//Storage Area Service
RegisterAlarm(Trigger := fbStorageArea.fbWarehouse.fbReloadBox.Error,				ID := GVL_ErrorCode.GC_ALARM_STO_RELOAD_BOX,value := E_Severity.Level4,Message := fbStorageArea.fbWarehouse.fbReloadBox.Status,			Category := 1);
RegisterAlarm(Trigger := fbStorageArea.fbWarehouse.fbFeedInBox.Error,				ID := GVL_ErrorCode.GC_ALARM_STO_FEEDIN_BOX,value := E_Severity.Level4,Message := fbStorageArea.fbWarehouse.fbFeedInBox.Status,			Category := 1);
RegisterAlarm(Trigger := fbStorageArea.fbAddBoxes.Error ,							ID := GVL_ErrorCode.GC_ALARM_STO_ADD_BOXES,value := E_Severity.Level4,Message := fbStorageArea.fbAddBoxes.Status,							Category := 1);
RegisterAlarm(Trigger := fbStorageArea.fbBoxSupplyCtrl.Error ,						ID := GVL_ErrorCode.GC_ALARM_STO_BOX_SUPPLY,value := E_Severity.Level4,Message := fbStorageArea.fbBoxSupplyCtrl.Status,					Category := 1);
RegisterAlarm(Trigger := fbStorageArea.fbFeedInEmptyBoxWithRobot.Error ,			ID := GVL_ErrorCode.GC_ALARM_STO_FEEDIN_EMPTY,value := E_Severity.Level4,Message := fbStorageArea.fbFeedInEmptyBoxWithRobot.Status,			Category := 1);
RegisterAlarm(Trigger := fbStorageArea.fbReloadRoundBeltBoxWithRobot.Error ,		ID := GVL_ErrorCode.GC_ALARM_STO_RELOAD_ROUNDBELT,value := E_Severity.Level4,Message := fbStorageArea.fbReloadRoundBeltBoxWithRobot.Status,		Category := 1);
RegisterAlarm(Trigger := fbStorageArea.fbRobotAbsMove.Error ,						ID := GVL_ErrorCode.GC_ALARM_STO_ROBOT_ABS_MOVE,value := E_Severity.Level4,Message := fbStorageArea.fbRobotAbsMove.Status,						Category := 1);
RegisterAlarm(Trigger := fbStorageArea.fbRobotRegionMove_AllocatedConveyor.Error ,	ID := GVL_ErrorCode.GC_ALARM_STO_REGION_ALLOC_CV,value := E_Severity.Level4,Message := fbStorageArea.fbRobotRegionMove_AllocatedConveyor.Status,Category := 1);
RegisterAlarm(Trigger := fbStorageArea.fbRobotRegionMove_BufferArea.Error ,			ID := GVL_ErrorCode.GC_ALARM_STO_REGION_BUFFER,value := E_Severity.Level4,Message := fbStorageArea.fbRobotRegionMove_BufferArea.Status,		Category := 1);
RegisterAlarm(Trigger := fbStorageArea.fbRobotRegionMove_FeedInConveyor.Error ,		ID := GVL_ErrorCode.GC_ALARM_STO_REGION_FEEDIN_CV,value := E_Severity.Level4,Message := fbStorageArea.fbRobotRegionMove_FeedInConveyor.Status,	Category := 1);
RegisterAlarm(Trigger := fbStorageArea.fbRobotRegionMove_PullOutConveyor.Error ,	ID := GVL_ErrorCode.GC_ALARM_STO_REGION_PULLOUT_CV,value := E_Severity.Level4,Message := fbStorageArea.fbRobotRegionMove_PullOutConveyor.Status,	Category := 1);
RegisterAlarm(Trigger := fbStorageArea.fbRobotRegionMove_RoundBelt.Error ,			ID := GVL_ErrorCode.GC_ALARM_STO_REGION_ROUNDBELT,value := E_Severity.Level4,Message := fbStorageArea.fbRobotRegionMove_RoundBelt.Status,		Category := 1);
RegisterAlarm(Trigger := fbStorageArea.fbUpperFeedInConveyor.Error ,				ID := GVL_ErrorCode.GC_ALARM_STO_UPPER_FEEDIN_CV,value := E_Severity.Level4,Message := fbStorageArea.fbUpperFeedInConveyor.Status,				Category := 1);
RegisterAlarm(Trigger := fbStorageArea.fbWareHouseWithRobotMove.Error ,				ID := GVL_ErrorCode.GC_ALARM_STO_WAREHOUSE_ROBOT,value := E_Severity.Level4,Message := fbStorageArea.fbWareHouseWithRobotMove.Status,			Category := 1);



//Storage Cabinet Internal Service
RegisterAlarm(Trigger := fbStorageArea.fbFeedInRoundBeltBoxToWareHouse.Error,		ID := GVL_ErrorCode.GC_ALARM_STO_FEEDIN_RB_TO_WH,value := E_Severity.Level3,Message := fbStorageArea.fbFeedInRoundBeltBoxToWareHouse.Status,Category := 1);
RegisterAlarm(Trigger := fbStorageArea._fbDaimeterMovement.Error,					ID := GVL_ErrorCode.GC_ALARM_STO_DIAMETER_MOVEMENT,value := E_Severity.Level3,Message := fbStorageArea._fbDaimeterMovement.Status,			Category := 1);
RegisterAlarm(Trigger := fbStorageArea.fbRobotSelfHoming.Error,						ID := GVL_ErrorCode.GC_ALARM_STO_ROBOTSELFHOMING,value := E_Severity.Level3,Message := fbStorageArea.fbRobotSelfHoming.Status,				Category := 1);
RegisterAlarm(Trigger := fbStorageArea.fbWareHouseInnerPickToRoundBelt.Error,		ID := GVL_ErrorCode.GC_AlARM_STO_ROBOTINNERPICK,value := E_Severity.Level3,Message := fbStorageArea.fbWareHouseInnerPickToRoundBelt.Status,	Category := 1);
RegisterAlarm(Trigger := fbStorageArea.fbWareHouseInnerPickToRoundBeltBatch.Error,  ID := GVL_ErrorCode.GC_AlARM_STO_ROBOTINNERPICK_BATCH,value := E_Severity.Level3,Message := fbStorageArea.fbWareHouseInnerPickToRoundBeltBatch.Status,	Category := 1);
RegisterAlarm(Trigger := fbStorageArea.fbFeedInRoundBeltBoxBatch.Error,  			ID := GVL_ErrorCode.GC_AlARM_STO_ROUNDBELTTOWAREHOUSE_BATCH,value := E_Severity.Level3,Message := fbStorageArea.fbFeedInRoundBeltBoxBatch.Status,	Category := 1);


//Allocate Area Service
RegisterAlarm(Trigger := fbAllocateArea.fb_AllocateBatchMode.Error ,				ID := GVL_ErrorCode.GC_ALARM_ALC_BATCH_MODE,value := E_Severity.Level3,Message := fbAllocateArea.fb_AllocateBatchMode.Status,			Category := 2);
RegisterAlarm(Trigger := fbAllocateArea.fb_AllocateBatchMode_Reverse.Error ,		ID := GVL_ErrorCode.GC_ALARM_ALC_BATCH_REVERSE,value := E_Severity.Level3,Message := fbAllocateArea.fb_AllocateBatchMode_Reverse.Status,	Category := 2);
RegisterAlarm(Trigger := fbAllocateArea.fbDifferentCVCamera.xError ,				ID := GVL_ErrorCode.GC_ALARM_ALC_DIFF_CV_CAMERA,value := E_Severity.Level3,Message := fbAllocateArea.fbDifferentCVCamera.ErrorMsg,			Category := 2);
RegisterAlarm(Trigger := fbAllocateArea.fbOutRobot_BoxMoveReverse.Error ,			ID := GVL_ErrorCode.GC_ALARM_ALC_OUTROBOT_REVERSE,value := E_Severity.Level3,Message := fbAllocateArea.fbOutRobot_BoxMoveReverse.Status,		Category := 2);
RegisterAlarm(Trigger := fbAllocateArea.fbOutRobot_EmptyBoxMove.Error ,				ID := GVL_ErrorCode.GC_ALARM_ALC_OUTROBOT_EMPTY,value := E_Severity.Level3,Message := fbAllocateArea.fbOutRobot_EmptyBoxMove.Status,		Category := 2);
RegisterAlarm(Trigger := fbAllocateArea.fbOutRobot_RareBoxMove.Error ,				ID := GVL_ErrorCode.GC_ALARM_ALC_OUTROBOT_RARE,value := E_Severity.Level3,Message := fbAllocateArea.fbOutRobot_RareBoxMove.Status,		Category := 2);
RegisterAlarm(Trigger := fbAllocateArea.fbPulloutCV.Error ,							ID := GVL_ErrorCode.GC_ALARM_ALC_PULLOUT_CV,value := E_Severity.Level3,Message := fbAllocateArea.fbPulloutCV.Status,					Category := 2);
RegisterAlarm(Trigger := fbAllocateArea.RoundBeltControl.xError ,					ID := GVL_ErrorCode.GC_ALARM_ALC_ROUNDBELT,value := E_Severity.Level3,Message := fbAllocateArea.RoundBeltControl.ErrorMsg,			Category := 2);
RegisterAlarm(Trigger := fbAllocateArea.fbSameSizeCVCamera.xError ,					ID := GVL_ErrorCode.GC_ALARM_ALC_SAME_CV_CAMERA,value := E_Severity.Level3,Message := fbAllocateArea.fbSameSizeCVCamera.ErrorMsg,			Category := 2);
RegisterAlarm(Trigger := fbAllocateArea.fbSameSizeCVCamera_Reverse.xError ,			ID := GVL_ErrorCode.GC_ALARM_ALC_SAME_CV_CAMERA_REVERSE,value := E_Severity.Level3,Message := fbAllocateArea.fbSameSizeCVCamera_Reverse.ErrorMsg,	Category := 2);
RegisterAlarm(Trigger := fbAllocateArea.TurnTableControl.xError ,					ID := GVL_ErrorCode.GC_ALARM_ALC_TURNTABLE,value := E_Severity.Level3,Message := fbAllocateArea.TurnTableControl.ErrorMsg,			Category := 2);
RegisterAlarm(Trigger := fbAllocateArea.fbOutRobot_TurnTableToRoundBelt.Error ,		ID := GVL_ErrorCode.GC_ALARM_ALC_OUTROBOT_TT_TO_RB,value := E_Severity.Level3,Message := fbAllocateArea.fbOutRobot_TurnTableToRoundBelt.Status,Category := 2);
RegisterAlarm(Trigger := fbAllocateArea.fbAllocateRobotNeedlingMove.xError, 		ID := GVL_ErrorCode.GC_ALARM_ALC_NEEDLING_MOVE,value:= E_Severity.Level3,Message:=fbAllocateArea.fbAllocateRobotNeedlingMove.ErrorMsg,				Category :=2);
RegisterAlarm(Trigger := fbAllocateArea.fbReverseBoxToWareHouse.Error, 				ID := GVL_ErrorCode.GC_ALARM_ALC_REVERSE_TO_WAREHOUSE,value:= E_Severity.Level3,Message	:= fbAllocateArea.fbReverseBoxToWareHouse.Status,		Category :=2);
RegisterAlarm(Trigger := fbAllocateArea.fbReverseBatchPickAndPhoto.Error, 			ID := GVL_ErrorCode.GC_ALARM_ALC_REVERSE_TO_WAREHOUSE_BATCH,value:= E_Severity.Level3,Message	:= fbAllocateArea.fbReverseBatchPickAndPhoto.Status,	Category :=2);



//Shipping Area Service
RegisterAlarm(Trigger := fbShippingArea.fbShippingRobot_Left.Error ,			ID := GVL_ErrorCode.GC_ALARM_SHP_ROBOT_LEFT,value := E_Severity.Level3,Message := fbShippingArea.fbShippingRobot_Left.Status,Category := 3);
RegisterAlarm(Trigger := fbShippingArea.fbShippingRobot_Right.Error ,			ID := GVL_ErrorCode.GC_ALARM_SHP_ROBOT_RIGHT,value := E_Severity.Level3,Message := fbShippingArea.fbShippingRobot_Right.Status,Category := 3);
RegisterAlarm(Trigger := fbShippingArea.fbShippingRobot_TransmitCVEnd.Error ,	ID := GVL_ErrorCode.GC_ALARM_SHP_ROBOT_TRANSMIT_END,value := E_Severity.Level3,Message := fbShippingArea.fbShippingRobot_TransmitCVEnd.Status,Category := 3);
RegisterAlarm(Trigger := fbShippingArea.fbShippingLeftSideTransCV.xError ,		ID := GVL_ErrorCode.GC_ALARM_SHP_LEFT_TRANS_CV,value := E_Severity.Level3,Message := fbShippingArea.fbShippingLeftSideTransCV.ErrorMsg,Category := 3);
RegisterAlarm(Trigger := fbShippingArea.fbShippingRightSideTransCV.xError ,		ID := GVL_ErrorCode.GC_ALARM_SHP_RIGHT_TRANS_CV,value := E_Severity.Level3,Message := fbShippingArea.fbShippingRightSideTransCV.ErrorMsg,Category := 3);
RegisterAlarm(Trigger := fbShippingArea.fbShippingRobot_Buffer.Error ,			ID := GVL_ErrorCode.GC_ALARM_SHP_ROBOT_BUFFER,value := E_Severity.Level3,Message := fbShippingArea.fbShippingRobot_Buffer.status,Category := 3);
RegisterAlarm(Trigger := fbShippingArea.fbShippingRobotTransfer.Error,			ID := GVL_ErrorCode.GC_ALARM_SHP_ROBOT_TRANSFER,value := E_Severity.Level3,Message := fbShippingArea.fbShippingRobotTransfer.Status,Category := 3);
RegisterAlarm(Trigger := fbShippingArea.fbShippingRobot_PhotoStandByPos.Error,	ID := GVL_ErrorCode.GC_ALARM_SHP_ROBOT_PHOTOSTANDBYPOS,value := E_Severity.Level3,Message := fbShippingArea.fbShippingRobot_PhotoStandByPos.Status,Category := 3);
RegisterAlarm(Trigger := fbShippingArea.fbShippingPlateScan.Error,				ID := GVL_ErrorCode.GC_ALARM_SHP_ROBOT_SCANPICK,value := E_Severity.Level3,Message := fbShippingArea.fbShippingPlateScan.Status,Category := 3);


// Cylinder Allocate Area component
RegisterAlarm(Trigger := Cylinder.List.fbAllocateRobot_LeftClamp1.xError,		ID := GVL_ErrorCode.GC_ALARM_CYL_ALC_ROBOT_LCLAMP1,value := E_Severity.Level2,Message := Cylinder.List.fbAllocateRobot_LeftClamp1.ErrorMsg,Category := 2);
RegisterAlarm(Trigger := Cylinder.List.fbAllocateRobot_LeftClamp2.xError,		ID := GVL_ErrorCode.GC_ALARM_CYL_ALC_ROBOT_LCLAMP2,value := E_Severity.Level2,Message := Cylinder.List.fbAllocateRobot_LeftClamp2.ErrorMsg,Category := 2);
RegisterAlarm(Trigger := Cylinder.List.fbAllocateRobot_LeftVert1.xError,		ID := GVL_ErrorCode.GC_ALARM_CYL_ALC_ROBOT_LVERT1,value := E_Severity.Level2,Message := Cylinder.List.fbAllocateRobot_LeftVert1.ErrorMsg,Category := 2);
RegisterAlarm(Trigger := Cylinder.List.fbAllocateRobot_LeftVert2.xError,		ID := GVL_ErrorCode.GC_ALARM_CYL_ALC_ROBOT_LVERT2,value := E_Severity.Level2,Message := Cylinder.List.fbAllocateRobot_LeftVert2.ErrorMsg,Category := 2);
RegisterAlarm(Trigger := Cylinder.List.fbAllocateRobot_RightClamp1.xError,		ID := GVL_ErrorCode.GC_ALARM_CYL_ALC_ROBOT_RCLAMP1,value := E_Severity.Level2,Message := Cylinder.List.fbAllocateRobot_RightClamp1.ErrorMsg,Category := 2);
RegisterAlarm(Trigger := Cylinder.List.fbAllocateRobot_RightClamp2.xError,		ID := GVL_ErrorCode.GC_ALARM_CYL_ALC_ROBOT_RCLAMP2,value := E_Severity.Level2,Message := Cylinder.List.fbAllocateRobot_RightClamp2.ErrorMsg,Category := 2);
RegisterAlarm(Trigger := Cylinder.List.fbAllocateRobot_RightVert1.xError,		ID := GVL_ErrorCode.GC_ALARM_CYL_ALC_ROBOT_RVERT1,value := E_Severity.Level2,Message := Cylinder.List.fbAllocateRobot_RightVert1.ErrorMsg,Category := 2);
RegisterAlarm(Trigger := Cylinder.List.fbAllocateRobot_RightVert2.xError,		ID := GVL_ErrorCode.GC_ALARM_CYL_ALC_ROBOT_RVERT2,value := E_Severity.Level2,Message := Cylinder.List.fbAllocateRobot_RightVert2.ErrorMsg,Category := 2);
RegisterAlarm(Trigger := Cylinder.List.fbRoundBelt_WorkZone_Press.xError,		ID := GVL_ErrorCode.GC_ALARM_CYL_ALC_RB_WORK_PRESS,value := E_Severity.Level2,Message := Cylinder.List.fbRoundBelt_WorkZone_Press.ErrorMsg,Category := 2);
RegisterAlarm(Trigger := Cylinder.List.fbRoundBelt_WorkZone_Plug.xError,		ID := GVL_ErrorCode.GC_ALARM_CYL_ALC_RB_WORK_PLUG,value := E_Severity.Level2,Message := Cylinder.List.fbRoundBelt_WorkZone_Plug.ErrorMsg,Category := 2);
RegisterAlarm(Trigger := Cylinder.List.fbRoundBelt_ChargeZone_Plug.xError,		ID := GVL_ErrorCode.GC_ALARM_CYL_ALC_RB_CHARGE_PLUG,value := E_Severity.Level2,Message := Cylinder.List.fbRoundBelt_ChargeZone_Plug.ErrorMsg,Category := 2);
RegisterAlarm(Trigger := Cylinder.List.fbRoundBelt_TransmitCVZone_Plug.xError,	ID := GVL_ErrorCode.GC_ALARM_CYL_ALC_RB_TRANS_PLUG,value := E_Severity.Level2,Message := Cylinder.List.fbRoundBelt_TransmitCVZone_Plug.ErrorMsg,Category := 2);
RegisterAlarm(Trigger := Cylinder.List.fbOutRobot_AsideVert.xError,				ID := GVL_ErrorCode.GC_ALARM_CYL_ALC_OUTROBOT_AVERT,value := E_Severity.Level2,Message := Cylinder.List.fbOutRobot_AsideVert.ErrorMsg,Category := 2);
RegisterAlarm(Trigger := Cylinder.List.fbOutRobot_BsideVert.xError,				ID := GVL_ErrorCode.GC_ALARM_CYL_ALC_OUTROBOT_BVERT,value := E_Severity.Level2,Message := Cylinder.List.fbOutRobot_BsideVert.ErrorMsg,Category := 2);
RegisterAlarm(Trigger := Cylinder.List.fbOutRobot_AsideClamp.xError,			ID := GVL_ErrorCode.GC_ALARM_CYL_ALC_OUTROBOT_ACLAMP,value := E_Severity.Level2,Message := Cylinder.List.fbOutRobot_AsideClamp.ErrorMsg,Category := 2);
RegisterAlarm(Trigger := Cylinder.List.fbOutRobot_BsideClamp.xError,			ID := GVL_ErrorCode.GC_ALARM_CYL_ALC_OUTROBOT_BCLAMP,value := E_Severity.Level2,Message := Cylinder.List.fbOutRobot_BsideClamp.ErrorMsg,Category := 2);
RegisterAlarm(Trigger := Cylinder.List.fbTransmitCV_CamaraHoriz.xError,			ID := GVL_ErrorCode.GC_ALARM_CYL_ALC_TRANS_CAMHORIZ,value := E_Severity.Level2,Message := Cylinder.List.fbTransmitCV_CamaraHoriz.ErrorMsg,Category := 2);
RegisterAlarm(Trigger := Cylinder.List.fbDifferentSizeCV_Press2.xError,			ID := GVL_ErrorCode.GC_ALARM_CYL_ALC_DIFF_PRESS2,value := E_Severity.Level2,Message := Cylinder.List.fbDifferentSizeCV_Press2.ErrorMsg,Category := 2);
RegisterAlarm(Trigger := Cylinder.List.fbDifferentSizeCV_Press1.xError,			ID := GVL_ErrorCode.GC_ALARM_CYL_ALC_DIFF_PRESS1,value := E_Severity.Level2,Message := Cylinder.List.fbDifferentSizeCV_Press1.ErrorMsg,Category := 2);
RegisterAlarm(Trigger := Cylinder.List.fbDifferentSizeCV_Block1.xError,			ID := GVL_ErrorCode.GC_ALARM_CYL_ALC_DIFF_BLOCK1_2,value := E_Severity.Level2,Message := Cylinder.List.fbDifferentSizeCV_Block1.ErrorMsg,Category := 2);
RegisterAlarm(Trigger := Cylinder.List.fbSameSizeCV_Press4.xError,				ID := GVL_ErrorCode.GC_ALARM_CYL_ALC_SAME_PRESS4,value := E_Severity.Level2,Message := Cylinder.List.fbSameSizeCV_Press4.ErrorMsg,Category := 2);
RegisterAlarm(Trigger := Cylinder.List.fbSameSizeCV_Press3.xError,				ID := GVL_ErrorCode.GC_ALARM_CYL_ALC_SAME_PRESS3,value := E_Severity.Level2,Message := Cylinder.List.fbSameSizeCV_Press3.ErrorMsg,Category := 2);
RegisterAlarm(Trigger := Cylinder.List.fbSameSizeCV_Press2.xError,				ID := GVL_ErrorCode.GC_ALARM_CYL_ALC_SAME_PRESS2,value := E_Severity.Level2,Message := Cylinder.List.fbSameSizeCV_Press2.ErrorMsg,Category := 2);
RegisterAlarm(Trigger := Cylinder.List.fbSameSizeCV_Press1.xError,				ID := GVL_ErrorCode.GC_ALARM_CYL_ALC_SAME_PRESS1,value := E_Severity.Level2,Message := Cylinder.List.fbSameSizeCV_Press1.ErrorMsg,Category := 2);
RegisterAlarm(Trigger := Cylinder.List.fbSameSizeCV_Block2.xError,				ID := GVL_ErrorCode.GC_ALARM_CYL_ALC_SAME_BLOCK2,value := E_Severity.Level2,Message := Cylinder.List.fbSameSizeCV_Block2.ErrorMsg,Category := 2);
RegisterAlarm(Trigger := Cylinder.List.fbSameSizeCV_Block1.xError,				ID := GVL_ErrorCode.GC_ALARM_CYL_ALC_SAME_BLOCK1,value := E_Severity.Level2,Message := Cylinder.List.fbSameSizeCV_Block1.ErrorMsg,Category := 2);
RegisterAlarm(Trigger := Cylinder.List.fbPullOutCV_AsidePress1.xError,			ID := GVL_ErrorCode.GC_ALARM_CYL_ALC_PULLOUT_APRESS1,value := E_Severity.Level2,Message := Cylinder.List.fbPullOutCV_AsidePress1.ErrorMsg,Category := 2);
RegisterAlarm(Trigger := Cylinder.List.fbPullOutCV_AsidePress2.xError,			ID := GVL_ErrorCode.GC_ALARM_CYL_ALC_PULLOUT_APRESS2,value := E_Severity.Level2,Message := Cylinder.List.fbPullOutCV_AsidePress2.ErrorMsg,Category := 2);
RegisterAlarm(Trigger := Cylinder.List.fbPullOutCV_AsideBlock.xError,			ID := GVL_ErrorCode.GC_ALARM_CYL_ALC_PULLOUT_ABLOCK,value := E_Severity.Level2,Message := Cylinder.List.fbPullOutCV_AsideBlock.ErrorMsg,Category := 2);
RegisterAlarm(Trigger := Cylinder.List.fbPullOutCV_BsidePress1.xError,			ID := GVL_ErrorCode.GC_ALARM_CYL_ALC_PULLOUT_BPRESS1,value := E_Severity.Level2,Message := Cylinder.List.fbPullOutCV_BsidePress1.ErrorMsg,Category := 2);
RegisterAlarm(Trigger := Cylinder.List.fbPullOutCV_BsidePress2.xError,			ID := GVL_ErrorCode.GC_ALARM_CYL_ALC_PULLOUT_BPRESS2,value := E_Severity.Level2,Message := Cylinder.List.fbPullOutCV_BsidePress2.ErrorMsg,Category := 2);
RegisterAlarm(Trigger := Cylinder.List.fbPullOutCV_BsideBlock.xError,			ID := GVL_ErrorCode.GC_ALARM_CYL_ALC_PULLOUT_BBLOCK,value := E_Severity.Level2,Message := Cylinder.List.fbPullOutCV_BsideBlock.ErrorMsg,Category := 2);

// Cyliner Storage Area component
RegisterAlarm(Trigger := Cylinder.List.fbUpCV_FeedInPress1.xError,				ID := GVL_ErrorCode.GC_ALARM_CYL_STO_UPCV_FEEDIN1,value := E_Severity.Level2,Message := Cylinder.List.fbUpCV_FeedInPress1.ErrorMsg,Category := 1);
RegisterAlarm(Trigger := Cylinder.List.fbUpCV_FeedInPress2.xError,				ID := GVL_ErrorCode.GC_ALARM_CYL_STO_UPCV_FEEDIN2,value := E_Severity.Level2,Message := Cylinder.List.fbUpCV_FeedInPress2.ErrorMsg,Category := 1);
RegisterAlarm(Trigger := Cylinder.List.fbUpCV_DiameterPress.xError,				ID := GVL_ErrorCode.GC_ALARM_CYL_STO_UPCV_DIAMETER,value := E_Severity.Level2,Message := Cylinder.List.fbUpCV_DiameterPress.ErrorMsg,Category := 1);
RegisterAlarm(Trigger := Cylinder.List.fbUpCV_CamaraPress1.xError,				ID := GVL_ErrorCode.GC_ALARM_CYL_STO_UPCV_CAM1,value := E_Severity.Level2,Message := Cylinder.List.fbUpCV_CamaraPress1.ErrorMsg,Category := 1);
RegisterAlarm(Trigger := Cylinder.List.fbUpCV_CamaraPress2.xError,				ID := GVL_ErrorCode.GC_ALARM_CYL_STO_UPCV_CAM2,value := E_Severity.Level2,Message := Cylinder.List.fbUpCV_CamaraPress2.ErrorMsg,Category := 1);
RegisterAlarm(Trigger := Cylinder.List.fbUpCV_CamaraPress3.xError,				ID := GVL_ErrorCode.GC_ALARM_CYL_STO_UPCV_CAM3,value := E_Severity.Level2,Message := Cylinder.List.fbUpCV_CamaraPress3.ErrorMsg,Category := 1);
RegisterAlarm(Trigger := Cylinder.List.fbUpCV_CamaraPress4.xError,				ID := GVL_ErrorCode.GC_ALARM_CYL_STO_UPCV_CAM4,value := E_Severity.Level2,Message := Cylinder.List.fbUpCV_CamaraPress4.ErrorMsg,Category := 1);
RegisterAlarm(Trigger := Cylinder.List.fbUpCV_Block1.xError,					ID := GVL_ErrorCode.GC_ALARM_CYL_STO_UPCV_BLOCK1,value := E_Severity.Level2,Message := Cylinder.List.fbUpCV_Block1.ErrorMsg,Category := 1);
RegisterAlarm(Trigger := Cylinder.List.fbUpCV_Block2.xError,					ID := GVL_ErrorCode.GC_ALARM_CYL_STO_UPCV_BLOCK2,value := E_Severity.Level2,Message := Cylinder.List.fbUpCV_Block2.ErrorMsg,Category := 1);
RegisterAlarm(Trigger := Cylinder.List.fbUpCV_Block3.xError,					ID := GVL_ErrorCode.GC_ALARM_CYL_STO_UPCV_BLOCK3,value := E_Severity.Level2,Message := Cylinder.List.fbUpCV_Block3.ErrorMsg,Category := 1);
RegisterAlarm(Trigger := Cylinder.List.fbUpCV_DiameterHoriz.xError,				ID := GVL_ErrorCode.GC_ALARM_CYL_STO_UPCV_DIA_HORIZ,value := E_Severity.Level2,Message := Cylinder.List.fbUpCV_DiameterHoriz.ErrorMsg,Category := 1);
RegisterAlarm(Trigger := Cylinder.List.fbUpCV_DiameterVert.xError,				ID := GVL_ErrorCode.GC_ALARM_CYL_STO_UPCV_DIA_VERT,value := E_Severity.Level2,Message := Cylinder.List.fbUpCV_DiameterVert.ErrorMsg,Category := 1);
RegisterAlarm(Trigger := Cylinder.List.fbUpCV_DiameterClamp.xError,				ID := GVL_ErrorCode.GC_ALARM_CYL_STO_UPCV_DIA_CLAMP,value := E_Severity.Level2,Message := Cylinder.List.fbUpCV_DiameterClamp.ErrorMsg,Category := 1);
RegisterAlarm(Trigger := Cylinder.List.fbStackPush.xError,						ID := GVL_ErrorCode.GC_ALARM_CYL_STO_STACK_PUSH,value := E_Severity.Level2,Message := Cylinder.List.fbStackPush.ErrorMsg,Category := 1);
RegisterAlarm(Trigger := Cylinder.List.fbLowCV_Press1.xError,					ID := GVL_ErrorCode.GC_ALARM_CYL_STO_LOWCV_PRESS1,value := E_Severity.Level2,Message := Cylinder.List.fbLowCV_Press1.ErrorMsg,Category := 1);
RegisterAlarm(Trigger := Cylinder.List.fbLowCV_Press2.xError,					ID := GVL_ErrorCode.GC_ALARM_CYL_STO_LOWCV_PRESS2,value := E_Severity.Level2,Message := Cylinder.List.fbLowCV_Press2.ErrorMsg,Category := 1);
RegisterAlarm(Trigger := Cylinder.List.fbLowCV_Press3.xError,					ID := GVL_ErrorCode.GC_ALARM_CYL_STO_LOWCV_PRESS3,value := E_Severity.Level2,Message := Cylinder.List.fbLowCV_Press3.ErrorMsg,Category := 1);
RegisterAlarm(Trigger := Cylinder.List.fbLowCV_Press4.xError,					ID := GVL_ErrorCode.GC_ALARM_CYL_STO_LOWCV_PRESS4,value := E_Severity.Level2,Message := Cylinder.List.fbLowCV_Press4.ErrorMsg,Category := 1);
RegisterAlarm(Trigger := Cylinder.List.fbLowCV_Block1.xError,					ID := GVL_ErrorCode.GC_ALARM_CYL_STO_LOWCV_BLOCK1,value := E_Severity.Level2,Message := Cylinder.List.fbLowCV_Block1.ErrorMsg,Category := 1);
RegisterAlarm(Trigger := Cylinder.List.fbLowCV_Block2.xError,					ID := GVL_ErrorCode.GC_ALARM_CYL_STO_LOWCV_BLOCK2,value := E_Severity.Level2,Message := Cylinder.List.fbLowCV_Block2.ErrorMsg,Category := 1);

	
// Robot Error
IF fbStorageArea.fbStorageHoming.Homed THEN
	bStorageRobotError := fanucrobot.List.StorageRobot.Error;
ELSE
	bStorageRobotError := FALSE;
END_IF
IF fbShippingArea.fbShippingHoming.Homed THEN
	bShippingRobotError := fanucrobot.List.ShippingRobot.Error;
ELSE
	bShippingRobotError := FALSE;
END_IF

RegisterAlarm(Trigger := bStorageRobotError,	ID := 158,value := E_Severity.Level5,Message := fanucrobot.List.StorageRobot.ErrMsg,Category:=1);
RegisterAlarm(Trigger := bShippingRobotError,	ID := 159,value := E_Severity.Level5,Message := fanucrobot.List.ShippingRobot.ErrMsg,Category:=1);


// =========================================================================
// Fanuc 大手臂 (StorageRobot) 細項 alarm 160-176
// 17 條 alarm 對應 FB_FanucRobot_Basic_V2 內所有 _Status 字串。
// trigger 寫法：先算到 bFanucStoTrig[N] (RegisterAlarm.Trigger 是 VAR_IN_OUT，不能塞表達式)
// =========================================================================
bFanucStoTrig[1]  := bStorageRobotError AND fanucrobot.List.StorageRobot.ErrMsg = GVL_ErrorCode.GC_MSG_0220; // Upper data Overload
RegisterAlarm(Trigger := bFanucStoTrig[1],  ID := 160, value := E_Severity.Level5, Message := GVL_ErrorCode.GC_MSG_0220, Category := 1);
bFanucStoTrig[2]  := bStorageRobotError AND fanucrobot.List.StorageRobot.ErrMsg = GVL_ErrorCode.GC_MSG_0208; // Jaw Sensor no Respond
RegisterAlarm(Trigger := bFanucStoTrig[2],  ID := 161, value := E_Severity.Level5, Message := GVL_ErrorCode.GC_MSG_0208, Category := 1);
bFanucStoTrig[3]  := bStorageRobotError AND fanucrobot.List.StorageRobot.ErrMsg = GVL_ErrorCode.GC_MSG_0221; // Vision fault
RegisterAlarm(Trigger := bFanucStoTrig[3],  ID := 162, value := E_Severity.Level5, Message := GVL_ErrorCode.GC_MSG_0221, Category := 1);
bFanucStoTrig[4]  := bStorageRobotError AND fanucrobot.List.StorageRobot.ErrMsg = GVL_ErrorCode.GC_MSG_0205; // Get but Has Sensor no Respond
RegisterAlarm(Trigger := bFanucStoTrig[4],  ID := 163, value := E_Severity.Level5, Message := GVL_ErrorCode.GC_MSG_0205, Category := 1);
bFanucStoTrig[5]  := bStorageRobotError AND fanucrobot.List.StorageRobot.ErrMsg = GVL_ErrorCode.GC_MSG_0206; // Get But Jaw Has
RegisterAlarm(Trigger := bFanucStoTrig[5],  ID := 164, value := E_Severity.Level5, Message := GVL_ErrorCode.GC_MSG_0206, Category := 1);
bFanucStoTrig[6]  := bStorageRobotError AND fanucrobot.List.StorageRobot.ErrMsg = GVL_ErrorCode.GC_MSG_0207; // illegal value in tool offset
RegisterAlarm(Trigger := bFanucStoTrig[6],  ID := 165, value := E_Severity.Level5, Message := GVL_ErrorCode.GC_MSG_0207, Category := 1);
bFanucStoTrig[7]  := bStorageRobotError AND fanucrobot.List.StorageRobot.ErrMsg = GVL_ErrorCode.GC_MSG_0209; // Laser detected
RegisterAlarm(Trigger := bFanucStoTrig[7],  ID := 166, value := E_Severity.Level5, Message := GVL_ErrorCode.GC_MSG_0209, Category := 1);
bFanucStoTrig[8]  := bStorageRobotError AND fanucrobot.List.StorageRobot.ErrMsg = GVL_ErrorCode.GC_MSG_0216; // Not in Home Pos
RegisterAlarm(Trigger := bFanucStoTrig[8],  ID := 167, value := E_Severity.Level5, Message := GVL_ErrorCode.GC_MSG_0216, Category := 1);
bFanucStoTrig[9]  := bStorageRobotError AND fanucrobot.List.StorageRobot.ErrMsg = GVL_ErrorCode.GC_MSG_0210; // Read All offset data failue
RegisterAlarm(Trigger := bFanucStoTrig[9],  ID := 168, value := E_Severity.Level5, Message := GVL_ErrorCode.GC_MSG_0210, Category := 1);
bFanucStoTrig[10] := bStorageRobotError AND fanucrobot.List.StorageRobot.ErrMsg = GVL_ErrorCode.GC_MSG_0211; // Retry too many times
RegisterAlarm(Trigger := bFanucStoTrig[10], ID := 169, value := E_Severity.Level5, Message := GVL_ErrorCode.GC_MSG_0211, Category := 1);
bFanucStoTrig[11] := bStorageRobotError AND fanucrobot.List.StorageRobot.ErrMsg = GVL_ErrorCode.GC_MSG_0212; // Robot Disconnect
RegisterAlarm(Trigger := bFanucStoTrig[11], ID := 170, value := E_Severity.Level5, Message := GVL_ErrorCode.GC_MSG_0212, Category := 1);
bFanucStoTrig[12] := bStorageRobotError AND fanucrobot.List.StorageRobot.ErrMsg = GVL_ErrorCode.GC_MSG_0213; // Battary alarm
RegisterAlarm(Trigger := bFanucStoTrig[12], ID := 171, value := E_Severity.Level5, Message := GVL_ErrorCode.GC_MSG_0213, Category := 1);
bFanucStoTrig[13] := bStorageRobotError AND fanucrobot.List.StorageRobot.ErrMsg = GVL_ErrorCode.GC_MSG_0214; // fatal alarm
RegisterAlarm(Trigger := bFanucStoTrig[13], ID := 172, value := E_Severity.Level5, Message := GVL_ErrorCode.GC_MSG_0214, Category := 1);
bFanucStoTrig[14] := bStorageRobotError AND fanucrobot.List.StorageRobot.ErrMsg = GVL_ErrorCode.GC_MSG_0215; // Halt State
RegisterAlarm(Trigger := bFanucStoTrig[14], ID := 173, value := E_Severity.Level5, Message := GVL_ErrorCode.GC_MSG_0215, Category := 1);
bFanucStoTrig[15] := bStorageRobotError AND fanucrobot.List.StorageRobot.ErrMsg = GVL_ErrorCode.GC_MSG_0217; // RSR1 error
RegisterAlarm(Trigger := bFanucStoTrig[15], ID := 174, value := E_Severity.Level5, Message := GVL_ErrorCode.GC_MSG_0217, Category := 1);
bFanucStoTrig[16] := bStorageRobotError AND fanucrobot.List.StorageRobot.ErrMsg = GVL_ErrorCode.GC_MSG_0218; // RSR3 error
RegisterAlarm(Trigger := bFanucStoTrig[16], ID := 175, value := E_Severity.Level5, Message := GVL_ErrorCode.GC_MSG_0218, Category := 1);
bFanucStoTrig[17] := bStorageRobotError AND fanucrobot.List.StorageRobot.ErrMsg = GVL_ErrorCode.GC_MSG_0219; // TP got control
RegisterAlarm(Trigger := bFanucStoTrig[17], ID := 176, value := E_Severity.Level5, Message := GVL_ErrorCode.GC_MSG_0219, Category := 1);

// =========================================================================
// Fanuc 小手臂 (ShippingRobot) 細項 alarm 180-196
// =========================================================================
bFanucShpTrig[1]  := bShippingRobotError AND fanucrobot.List.ShippingRobot.ErrMsg = GVL_ErrorCode.GC_MSG_0220; // Upper data Overload
RegisterAlarm(Trigger := bFanucShpTrig[1],  ID := 180, value := E_Severity.Level5, Message := GVL_ErrorCode.GC_MSG_0220, Category := 1);
bFanucShpTrig[2]  := bShippingRobotError AND fanucrobot.List.ShippingRobot.ErrMsg = GVL_ErrorCode.GC_MSG_0208; // Jaw Sensor no Respond
RegisterAlarm(Trigger := bFanucShpTrig[2],  ID := 181, value := E_Severity.Level5, Message := GVL_ErrorCode.GC_MSG_0208, Category := 1);
bFanucShpTrig[3]  := bShippingRobotError AND fanucrobot.List.ShippingRobot.ErrMsg = GVL_ErrorCode.GC_MSG_0221; // Vision fault
RegisterAlarm(Trigger := bFanucShpTrig[3],  ID := 182, value := E_Severity.Level5, Message := GVL_ErrorCode.GC_MSG_0221, Category := 1);
bFanucShpTrig[4]  := bShippingRobotError AND fanucrobot.List.ShippingRobot.ErrMsg = GVL_ErrorCode.GC_MSG_0205; // Get but Has Sensor no Respond
RegisterAlarm(Trigger := bFanucShpTrig[4],  ID := 183, value := E_Severity.Level5, Message := GVL_ErrorCode.GC_MSG_0205, Category := 1);
bFanucShpTrig[5]  := bShippingRobotError AND fanucrobot.List.ShippingRobot.ErrMsg = GVL_ErrorCode.GC_MSG_0206; // Get But Jaw Has
RegisterAlarm(Trigger := bFanucShpTrig[5],  ID := 184, value := E_Severity.Level5, Message := GVL_ErrorCode.GC_MSG_0206, Category := 1);
bFanucShpTrig[6]  := bShippingRobotError AND fanucrobot.List.ShippingRobot.ErrMsg = GVL_ErrorCode.GC_MSG_0207; // illegal value in tool offset
RegisterAlarm(Trigger := bFanucShpTrig[6],  ID := 185, value := E_Severity.Level5, Message := GVL_ErrorCode.GC_MSG_0207, Category := 1);
bFanucShpTrig[7]  := bShippingRobotError AND fanucrobot.List.ShippingRobot.ErrMsg = GVL_ErrorCode.GC_MSG_0209; // Laser detected
RegisterAlarm(Trigger := bFanucShpTrig[7],  ID := 186, value := E_Severity.Level5, Message := GVL_ErrorCode.GC_MSG_0209, Category := 1);
bFanucShpTrig[8]  := bShippingRobotError AND fanucrobot.List.ShippingRobot.ErrMsg = GVL_ErrorCode.GC_MSG_0216; // Not in Home Pos
RegisterAlarm(Trigger := bFanucShpTrig[8],  ID := 187, value := E_Severity.Level5, Message := GVL_ErrorCode.GC_MSG_0216, Category := 1);
bFanucShpTrig[9]  := bShippingRobotError AND fanucrobot.List.ShippingRobot.ErrMsg = GVL_ErrorCode.GC_MSG_0210; // Read All offset data failue
RegisterAlarm(Trigger := bFanucShpTrig[9],  ID := 188, value := E_Severity.Level5, Message := GVL_ErrorCode.GC_MSG_0210, Category := 1);
bFanucShpTrig[10] := bShippingRobotError AND fanucrobot.List.ShippingRobot.ErrMsg = GVL_ErrorCode.GC_MSG_0211; // Retry too many times
RegisterAlarm(Trigger := bFanucShpTrig[10], ID := 189, value := E_Severity.Level5, Message := GVL_ErrorCode.GC_MSG_0211, Category := 1);
bFanucShpTrig[11] := bShippingRobotError AND fanucrobot.List.ShippingRobot.ErrMsg = GVL_ErrorCode.GC_MSG_0212; // Robot Disconnect
RegisterAlarm(Trigger := bFanucShpTrig[11], ID := 190, value := E_Severity.Level5, Message := GVL_ErrorCode.GC_MSG_0212, Category := 1);
bFanucShpTrig[12] := bShippingRobotError AND fanucrobot.List.ShippingRobot.ErrMsg = GVL_ErrorCode.GC_MSG_0213; // Battary alarm
RegisterAlarm(Trigger := bFanucShpTrig[12], ID := 191, value := E_Severity.Level5, Message := GVL_ErrorCode.GC_MSG_0213, Category := 1);
bFanucShpTrig[13] := bShippingRobotError AND fanucrobot.List.ShippingRobot.ErrMsg = GVL_ErrorCode.GC_MSG_0214; // fatal alarm
RegisterAlarm(Trigger := bFanucShpTrig[13], ID := 192, value := E_Severity.Level5, Message := GVL_ErrorCode.GC_MSG_0214, Category := 1);
bFanucShpTrig[14] := bShippingRobotError AND fanucrobot.List.ShippingRobot.ErrMsg = GVL_ErrorCode.GC_MSG_0215; // Halt State
RegisterAlarm(Trigger := bFanucShpTrig[14], ID := 193, value := E_Severity.Level5, Message := GVL_ErrorCode.GC_MSG_0215, Category := 1);
bFanucShpTrig[15] := bShippingRobotError AND fanucrobot.List.ShippingRobot.ErrMsg = GVL_ErrorCode.GC_MSG_0217; // RSR1 error
RegisterAlarm(Trigger := bFanucShpTrig[15], ID := 194, value := E_Severity.Level5, Message := GVL_ErrorCode.GC_MSG_0217, Category := 1);
bFanucShpTrig[16] := bShippingRobotError AND fanucrobot.List.ShippingRobot.ErrMsg = GVL_ErrorCode.GC_MSG_0218; // RSR3 error
RegisterAlarm(Trigger := bFanucShpTrig[16], ID := 195, value := E_Severity.Level5, Message := GVL_ErrorCode.GC_MSG_0218, Category := 1);
bFanucShpTrig[17] := bShippingRobotError AND fanucrobot.List.ShippingRobot.ErrMsg = GVL_ErrorCode.GC_MSG_0219; // TP got control
RegisterAlarm(Trigger := bFanucShpTrig[17], ID := 196, value := E_Severity.Level5, Message := GVL_ErrorCode.GC_MSG_0219, Category := 1);


// Servo Error
RegisterAlarm(Trigger := arAxisCtrl_gb[AxisNo.TurnTable].Admin.Axis.Status.Error,ID := GVL_ErrorCode.GC_ALARM_AXIS_TURNTABLE,value := E_Severity.Level6,Message := GVL_ErrorCode.GC_MSG_0181,Category := 2);
RegisterAlarm(Trigger := arAxisCtrl_gb[AxisNo.RoundBelt].Admin.Axis.Status.Error,ID := GVL_ErrorCode.GC_ALARM_AXIS_ROUNDBELT,value := E_Severity.Level6,Message := GVL_ErrorCode.GC_MSG_0182,Category := 2);
RegisterAlarm(Trigger := arAxisCtrl_gb[AxisNo.Allocate_X].Admin.Axis.Status.Error,ID := GVL_ErrorCode.GC_ALARM_AXIS_ALLOCATE_X,value := E_Severity.Level6,Message := GVL_ErrorCode.GC_MSG_0183,Category := 2);
RegisterAlarm(Trigger := arAxisCtrl_gb[AxisNo.Allocate_Y].Admin.Axis.Status.Error,ID := GVL_ErrorCode.GC_ALARM_AXIS_ALLOCATE_Y,value := E_Severity.Level6,Message := GVL_ErrorCode.GC_MSG_0184,Category := 2);
RegisterAlarm(Trigger := arAxisCtrl_gb[AxisNo.OutRobot_X].Admin.Axis.Status.Error,ID := GVL_ErrorCode.GC_ALARM_AXIS_OUTROBOT_X,value := E_Severity.Level6,Message := GVL_ErrorCode.GC_MSG_0185,Category := 2);
RegisterAlarm(Trigger := arAxisCtrl_gb[AxisNo.OutRobot_Y].Admin.Axis.Status.Error,ID := GVL_ErrorCode.GC_ALARM_AXIS_OUTROBOT_Y,value := E_Severity.Level6,Message := GVL_ErrorCode.GC_MSG_0186,Category := 2);
RegisterAlarm(Trigger := arAxisCtrl_gb[AxisNo.RackMotor].Admin.Axis.Status.Error,ID := GVL_ErrorCode.GC_ALARM_AXIS_RACKMOTOR,value := E_Severity.Level6,Message := GVL_ErrorCode.GC_MSG_0187,Category := 1);

// ModbusRTU
// AND NOT stModbusByPassInternal.switchOff_N: power cycle 期間 (fbRebootModbusDevice
// step 0~500) 我們自己關了電源,bError 是預期的不應再爆 alarm。step 500 結束後
// stModbusByPassInternal 清回 FALSE,這時才恢復檢查 bError — 若還是 TRUE 表示
// 光電板真的壞了,alarm 才重新出現。
bByPassModBusRTU[1] := MAIN2_RS485.RS485_V2[1].bError AND NOT GVL_HMI.Setup.Mechanical.stModbusByPass.switchOff_1 AND NOT GVL_Machine.stModbusByPassInternal.switchOff_1;
bByPassModBusRTU[2] := MAIN2_RS485.RS485_V2[2].bError AND NOT GVL_HMI.Setup.Mechanical.stModbusByPass.switchOff_2 AND NOT GVL_Machine.stModbusByPassInternal.switchOff_2;
bByPassModBusRTU[3] := MAIN2_RS485.RS485_V2[3].bError AND NOT GVL_HMI.Setup.Mechanical.stModbusByPass.switchOff_3 AND NOT GVL_Machine.stModbusByPassInternal.switchOff_3;
bByPassModBusRTU[4] := MAIN2_RS485.RS485_V2[4].bError AND NOT GVL_HMI.Setup.Mechanical.stModbusByPass.switchOff_4 AND NOT GVL_Machine.stModbusByPassInternal.switchOff_4;

RegisterAlarm(Trigger := bByPassModBusRTU[1],ID := GVL_ErrorCode.GC_ALARM_MODBUSRTU	+ 1,value := E_Severity.Level2,Message := MAIN2_RS485.RS485_V2[1].ErrorMsg,Category := 1);
RegisterAlarm(Trigger := bByPassModBusRTU[2],ID := GVL_ErrorCode.GC_ALARM_MODBUSRTU + 2,value := E_Severity.Level2,Message := MAIN2_RS485.RS485_V2[2].ErrorMsg,Category := 1);
RegisterAlarm(Trigger := bByPassModBusRTU[3],ID := GVL_ErrorCode.GC_ALARM_MODBUSRTU + 3,value := E_Severity.Level2,Message := MAIN2_RS485.RS485_V2[3].ErrorMsg,Category := 1);
RegisterAlarm(Trigger := bByPassModBusRTU[4],ID := GVL_ErrorCode.GC_ALARM_MODBUSRTU + 4,value := E_Severity.Level2,Message := MAIN2_RS485.RS485_V2[4].ErrorMsg,Category := 1);





//Safe Door
IF NOT GVL_HMI.Setup.Mechanical.stSafetyByPass.SafeDoorByPass THEN
	SafeDoorsOpen[1] 	:=  NOT INPUT.bSafetyDoor1   AND NOT GVL_HMI.Setup.Mechanical.stSafetyByPass.SafeDoorByPass;	 
	SafeDoorsOpen[2] 	:=  NOT INPUT.bSafetyDoor2   AND NOT GVL_HMI.Setup.Mechanical.stSafetyByPass.SafeDoorByPass;	 
	SafeDoorsOpen[3] 	:=  NOT INPUT.bSafetyDoor3   AND NOT GVL_HMI.Setup.Mechanical.stSafetyByPass.SafeDoorByPass;	 
	SafeDoorsOpen[4] 	:=  NOT INPUT.bSafetyDoor4   AND NOT GVL_HMI.Setup.Mechanical.stSafetyByPass.SafeDoorByPass;
	SafeDoorsOpen[5] 	:=  NOT INPUT.bSafetyDoor5   AND NOT GVL_HMI.Setup.Mechanical.stSafetyByPass.SafeDoorByPass;	 
	SafeDoorsOpen[6] 	:=  NOT INPUT.bSafetyDoor6   AND NOT GVL_HMI.Setup.Mechanical.stSafetyByPass.SafeDoorByPass;	 
	SafeDoorsOpen[7] 	:=  NOT INPUT.bSafetyDoor7   AND NOT GVL_HMI.Setup.Mechanical.stSafetyByPass.SafeDoorByPass;	 
	SafeDoorsOpen[8] 	:=  NOT INPUT.bSafetyDoor8   AND NOT GVL_HMI.Setup.Mechanical.stSafetyByPass.SafeDoorByPass;	 
	SafeDoorsOpen[9] 	:=  NOT INPUT.bSafetyDoor9   AND NOT GVL_HMI.Setup.Mechanical.stSafetyByPass.SafeDoorByPass;	 
	SafeDoorsOpen[10] 	:=  NOT INPUT.bSafetyDoor10   AND NOT GVL_HMI.Setup.Mechanical.stSafetyByPass.SafeDoorByPass;	 
	SafeDoorsOpen[11] 	:=  NOT INPUT.bSafetyDoor11   AND NOT GVL_HMI.Setup.Mechanical.stSafetyByPass.SafeDoorByPass;	 
	SafeDoorsOpen[12] 	:=  NOT INPUT.bSafetyDoor12   AND NOT GVL_HMI.Setup.Mechanical.stSafetyByPass.SafeDoorByPass;	 
	SafeDoorsOpen[13] 	:=  NOT INPUT.bSafetyDoor13   AND NOT GVL_HMI.Setup.Mechanical.stSafetyByPass.SafeDoorByPass;	 
	SafeDoorsOpen[14] 	:=  NOT INPUT.bSafetyDoor14   AND NOT GVL_HMI.Setup.Mechanical.stSafetyByPass.SafeDoorByPass;	 
	SafeDoorsOpen[15] 	:=  NOT INPUT.bAllocate_Electrical_Cabinet_SafetyDoor   AND NOT GVL_HMI.Setup.Mechanical.stSafetyByPass.SafeDoorByPass;	 
	SafeDoorsOpen[16] 	:=  NOT INPUT.bShippingRobot_ElectricalCabinet_SafetyDoor   AND NOT GVL_HMI.Setup.Mechanical.stSafetyByPass.SafeDoorByPass;	 
ELSE
	FOR i := 1 TO 20 DO 
		SafeDoorsOpen[i] := FALSE;
	END_FOR
END_IF

	RegisterAlarm(Trigger := SafeDoorsOpen[1],  ID := GVL_ErrorCode.GC_ALARM_SAFE_DOOR_BASE + 1, value := E_Severity.Level2, Message := GVL_ErrorCode.GC_MSG_0188,  Category := 1);
	RegisterAlarm(Trigger := SafeDoorsOpen[2],  ID := GVL_ErrorCode.GC_ALARM_SAFE_DOOR_BASE + 2, value := E_Severity.Level2, Message := GVL_ErrorCode.GC_MSG_0189,  Category := 1);
	RegisterAlarm(Trigger := SafeDoorsOpen[3],  ID := GVL_ErrorCode.GC_ALARM_SAFE_DOOR_BASE + 3, value := E_Severity.Level2, Message := GVL_ErrorCode.GC_MSG_0190,  Category := 1);
	RegisterAlarm(Trigger := SafeDoorsOpen[4],  ID := GVL_ErrorCode.GC_ALARM_SAFE_DOOR_BASE + 4, value := E_Severity.Level2, Message := GVL_ErrorCode.GC_MSG_0191,  Category := 1);
	RegisterAlarm(Trigger := SafeDoorsOpen[5],  ID := GVL_ErrorCode.GC_ALARM_SAFE_DOOR_BASE + 5, value := E_Severity.Level2, Message := GVL_ErrorCode.GC_MSG_0192,  Category := 1);
	RegisterAlarm(Trigger := SafeDoorsOpen[6],  ID := GVL_ErrorCode.GC_ALARM_SAFE_DOOR_BASE + 6, value := E_Severity.Level2, Message := GVL_ErrorCode.GC_MSG_0193,  Category := 1);
	RegisterAlarm(Trigger := SafeDoorsOpen[7],  ID := GVL_ErrorCode.GC_ALARM_SAFE_DOOR_BASE + 7, value := E_Severity.Level2, Message := GVL_ErrorCode.GC_MSG_0194,  Category := 1);
	RegisterAlarm(Trigger := SafeDoorsOpen[8],  ID := GVL_ErrorCode.GC_ALARM_SAFE_DOOR_BASE + 8, value := E_Severity.Level2, Message := GVL_ErrorCode.GC_MSG_0195,  Category := 1);
	RegisterAlarm(Trigger := SafeDoorsOpen[9],	ID := GVL_ErrorCode.GC_ALARM_SAFE_DOOR_BASE + 9, value := E_Severity.Level2, Message := GVL_ErrorCode.GC_MSG_0196,  Category := 1);
	RegisterAlarm(Trigger := SafeDoorsOpen[10],	ID := GVL_ErrorCode.GC_ALARM_SAFE_DOOR_BASE + 10, value := E_Severity.Level2, Message := GVL_ErrorCode.GC_MSG_0197,  Category := 1);
	RegisterAlarm(Trigger := SafeDoorsOpen[11],	ID := GVL_ErrorCode.GC_ALARM_SAFE_DOOR_BASE + 11, value := E_Severity.Level2, Message := GVL_ErrorCode.GC_MSG_0198,  Category := 1);
	RegisterAlarm(Trigger := SafeDoorsOpen[12],	ID := GVL_ErrorCode.GC_ALARM_SAFE_DOOR_BASE + 12, value := E_Severity.Level2, Message := GVL_ErrorCode.GC_MSG_0199,  Category := 1);
	RegisterAlarm(Trigger := SafeDoorsOpen[13],	ID := GVL_ErrorCode.GC_ALARM_SAFE_DOOR_BASE + 13, value := E_Severity.Level2, Message := GVL_ErrorCode.GC_MSG_0200,  Category := 1);
	RegisterAlarm(Trigger := SafeDoorsOpen[14],	ID := GVL_ErrorCode.GC_ALARM_SAFE_DOOR_BASE + 14, value := E_Severity.Level2, Message := GVL_ErrorCode.GC_MSG_0201,  Category := 1);
	RegisterAlarm(Trigger := SafeDoorsOpen[15],	ID := GVL_ErrorCode.GC_ALARM_SAFE_DOOR_BASE + 15, value := E_Severity.Level2, Message := GVL_ErrorCode.GC_MSG_0202,  Category := 1);
	RegisterAlarm(Trigger := SafeDoorsOpen[16],	ID := GVL_ErrorCode.GC_ALARM_SAFE_DOOR_BASE + 16, value := E_Severity.Level2, Message := GVL_ErrorCode.GC_MSG_0203,  Category := 1); 


M_General_AlarmRegister := TRUE;
END_METHOD

METHOD M_GetCylinderError : BOOL
VAR_INPUT
END_VAR
VAR
	udiCylinderIndex : UDINT;
END_VAR
FOR udiCylinderIndex := 1 TO udiMax_CylinderNum DO
	IF Cylinder.arCylinder[udiCylinderIndex].xError THEN
		M_GetCylinderError := TRUE;
	END_IF
END_FOR
END_METHOD

METHOD M_HalfAuto_TableMove
VAR_INPUT
END_VAR
// TableMove service 
TableMove(
	xDone=> AllocateHalfAutoCommand.TableMove.Status.Done, 
	xBusy=> AllocateHalfAutoCommand.TableMove.Status.Busy, 
	xError=> AllocateHalfAutoCommand.TableMove.Status.Error, 
	xExecute:= AllocateHalfAutoCommand.TableMove.Ctrl.Execute, 
	xAbort:= AllocateHalfAutoCommand.TableMove.Ctrl.Abort,
	xReset :=  AllocateHalfAutoCommand.TableMove.Ctrl.Reset,
	Index:= AllocateHalfAutoCommand.TableMove.Ctrl.Index, 
	CurrentData:= CurrentData, 
	xAborted=> AllocateHalfAutoCommand.TableMove.Status.Aborted);
END_METHOD

METHOD M_Held
M_StateComplete();
END_METHOD

METHOD M_Holding
M_StateComplete();
END_METHOD

METHOD M_Idle
IF eModeCurrent = E_UnitMode.Auto THEN
	GVL_Machine.PackTags[UnitNo.Storage].Command.UnitMode := E_UnitMode.Auto;
	GVL_Machine.PackTags[UnitNo.Allocate].Command.UnitMode := E_UnitMode.Auto;
	GVL_Machine.PackTags[UnitNo.Shipping].Command.UnitMode := E_UnitMode.Auto;
ELSIF eModeCurrent = E_UnitMode.Manual THEN
	GVL_Machine.PackTags[UnitNo.Storage].Command.UnitMode := E_UnitMode.Manual;
	GVL_Machine.PackTags[UnitNo.Allocate].Command.UnitMode := E_UnitMode.Manual;
	GVL_Machine.PackTags[UnitNo.Shipping].Command.UnitMode := E_UnitMode.Manual;
END_IF

M_StateComplete();
END_METHOD

METHOD M_MachineHoming : BOOL
VAR_INPUT
END_VAR
fbMachineHoming.xExecute :=   Service_Handshake.MachineHome.HandShake.Execute;
fbMachineHoming.xAbort := Machine_Stop;

Service_Handshake.MachineHome.HandShake.Done := fbMachineHoming.xDone;
Service_Handshake.MachineHome.HandShake.Busy := fbMachineHoming.xBusy;
Service_Handshake.MachineHome.HandShake.Error := fbMachineHoming.xError;
END_METHOD

METHOD PRIVATE M_Manual_Axes
VAR_INPUT
END_VAR

VAR_INST
	AllowAllocateRobotMove : BOOL;
	AllowOutRobotMove : BOOL;
	AllowRoundBeltMove : BOOL;
	AllowTurnTable		:BOOL;
	AllowRackMotor		:BOOL;
END_VAR
// Safe check
AllowAllocateRobotMove := Cylinder.List.fbAllocateRobot_LeftVert1.InRearPosition AND
    Cylinder.List.fbAllocateRobot_LeftVert2.InRearPosition AND
    Cylinder.List.fbAllocateRobot_RightVert1.InRearPosition AND
    Cylinder.List.fbAllocateRobot_RightVert2.InRearPosition;

AllowOutRobotMove := Cylinder.List.fbOutRobot_AsideVert.InRearPosition AND Cylinder.List.fbOutRobot_BsideVert.InRearPosition;
AllowRoundBeltMove := Cylinder.List.fbRoundBelt_ChargeZone_Plug.InRearPosition AND
    Cylinder.List.fbRoundBelt_TransmitCVZone_Plug.InRearPosition AND
    Cylinder.List.fbRoundBelt_WorkZone_Plug.InRearPosition AND
    Cylinder.List.fbRoundBelt_WorkZone_Press.InRearPosition AND
    AllowAllocateRobotMove AND
    AllowOutRobotMove 
	AND NOT FanucRobot.List.StorageRobot.BZoneInWork AND NOT FanucRobot.List.StorageRobot.Bzone_AllowWork;

AllowTurnTable := Cylinder.List.fbTurntable_Press.InRearPosition;
AllowRackMotor := Cylinder.List.fbStackPush.InRearPosition;

// Axis controll
{region "AllocateRobot AxisX"}

IF AllocateManualCommand.AllocatedRobot.AxisX.JOG.MoveFWD AND AllowAllocateRobotMove  THEN
    arAxisCtrl_gb[AxisNo.Allocate_X].VelMode.Acc := CurrentData.Axes.Allocate_X.Manual.JogAcceleration;
    arAxisCtrl_gb[AxisNo.Allocate_X].VelMode.Dec := CurrentData.Axes.Allocate_X.Manual.JogDeceleration;
    arAxisCtrl_gb[AxisNo.Allocate_X].VelMode.Jerk := CurrentData.Axes.Allocate_X.Manual.JogJerk;
    arAxisCtrl_gb[AxisNo.Allocate_X].VelMode.Velocity := CurrentData.Axes.Allocate_X.Manual.JogVelocity;
    arAxisCtrl_gb[AxisNo.Allocate_X].Admin._OpMode.en := E_AXIS_MODE.ModeVel;
ELSIF AllocateManualCommand.AllocatedRobot.AxisX.JOG.MoveBWD AND AllowAllocateRobotMove THEN
    arAxisCtrl_gb[AxisNo.Allocate_X].VelMode.Acc := CurrentData.Axes.Allocate_X.Manual.JogAcceleration;
    arAxisCtrl_gb[AxisNo.Allocate_X].VelMode.Dec := CurrentData.Axes.Allocate_X.Manual.JogDeceleration;
    arAxisCtrl_gb[AxisNo.Allocate_X].VelMode.Jerk := CurrentData.Axes.Allocate_X.Manual.JogJerk;
    arAxisCtrl_gb[AxisNo.Allocate_X].VelMode.Velocity := CurrentData.Axes.Allocate_X.Manual.JogVelocity * -1;
    arAxisCtrl_gb[AxisNo.Allocate_X].Admin._OpMode.en := E_AXIS_MODE.ModeVel;
ELSIF AllocateManualCommand.AllocatedRobot.AxisX.PTP.Enable  AND AllowAllocateRobotMove THEN
    arAxisCtrl_gb[AxisNo.Allocate_X].PosMode.Acc := CurrentData.Axes.Allocate_X.Manual.PtpAcceleration;
    arAxisCtrl_gb[AxisNo.Allocate_X].PosMode.Dec := CurrentData.Axes.Allocate_X.Manual.PtpDeceleration;
    arAxisCtrl_gb[AxisNo.Allocate_X].PosMode.Jerk := CurrentData.Axes.Allocate_X.Manual.PtpJerk;
    arAxisCtrl_gb[AxisNo.Allocate_X].PosMode.Velocity := CurrentData.Axes.Allocate_X.Manual.PtpVelocity;
    arAxisCtrl_gb[AxisNo.Allocate_X].PosMode.Position := CurrentData.Axes.Allocate_X.Manual.PtpPosition;
    arAxisCtrl_gb[AxisNo.Allocate_X].Admin._OpMode.en := ModePosAbs;
ELSIF (AllocateManualCommand.AllocatedRobot.AxisX.Homing.Execute OR  fbAllocateArea.fbAllocateHome.AxisHomingRequest)  AND AllowAllocateRobotMove THEN
    arAxisCtrl_gb[AxisNo.Allocate_X].SetupMode.eHomingMode := E_HomingMode._17_Neg_LimitOutterRight;
    arAxisCtrl_gb[AxisNo.Allocate_X].SetupMode.FastVelo := CurrentData.Axes.Allocate_X.Homing.FastVelo;
    arAxisCtrl_gb[AxisNo.Allocate_X].SetupMode.SlowVelo := CurrentData.Axes.Allocate_X.Homing.SlowVelo;
    arAxisCtrl_gb[AxisNo.Allocate_X].SetupMode.lrOffset := CurrentData.Axes.Allocate_X.Homing.Offset;
    arAxisCtrl_gb[AxisNo.Allocate_X].SetupMode.lrSetPosition := CurrentData.Axes.Allocate_X.Homing.SetAbsolutePosition;
    arAxisCtrl_gb[AxisNo.Allocate_X].SetupMode.stPosBiasParameter.bSetPostionBias := TRUE;
    arAxisCtrl_gb[AxisNo.Allocate_X].Admin._OpMode.en := ModeHoming;
ELSIF TableMove.xBusy AND AllowAllocateRobotMove THEN
    arAxisCtrl_gb[AxisNo.Allocate_X].Admin._OpMode.en := ModePosAbs;
ELSIF fbAllocateArea.fbAllocateRobotNeedlingMove.xBusy AND AllowAllocateRobotMove THEN
	arAxisCtrl_gb[AxisNo.Allocate_X].PosMode.Acc := CurrentData.Axes.Allocate_X.Manual.PtpAcceleration;
    arAxisCtrl_gb[AxisNo.Allocate_X].PosMode.Dec := CurrentData.Axes.Allocate_X.Manual.PtpDeceleration;
    arAxisCtrl_gb[AxisNo.Allocate_X].PosMode.Jerk := CurrentData.Axes.Allocate_X.Manual.PtpJerk;
    arAxisCtrl_gb[AxisNo.Allocate_X].PosMode.Velocity := CurrentData.Axes.Allocate_X.Manual.PtpVelocity;
    arAxisCtrl_gb[AxisNo.Allocate_X].Admin._OpMode.en := ModePosAbs;	
  
ELSIF fbAllocateArea.fb_AllocateBatchMode.Busy AND AllowAllocateRobotMove THEN
    arAxisCtrl_gb[AxisNo.Allocate_X].Admin._OpMode.en := ModePosAbs;

					  
ELSE
    arAxisCtrl_gb[AxisNo.Allocate_X].Admin.StopDeceleration := 1000;
    arAxisCtrl_gb[AxisNo.Allocate_X].Admin._OpMode.en := E_AXIS_MODE.ModeAH;
		 
			 
END_IF
{endregion}

{region "AllocateRobot AxisY"}
IF AllocateManualCommand.AllocatedRobot.AxisY.JOG.MoveFWD AND AllowAllocateRobotMove THEN
    arAxisCtrl_gb[AxisNo.Allocate_Y].VelMode.Acc := CurrentData.Axes.Allocate_Y.Manual.JogAcceleration;
    arAxisCtrl_gb[AxisNo.Allocate_Y].VelMode.Dec := CurrentData.Axes.Allocate_Y.Manual.JogDeceleration;
    arAxisCtrl_gb[AxisNo.Allocate_Y].VelMode.Jerk := CurrentData.Axes.Allocate_Y.Manual.JogJerk;
    arAxisCtrl_gb[AxisNo.Allocate_Y].VelMode.Velocity := CurrentData.Axes.Allocate_Y.Manual.JogVelocity;
    arAxisCtrl_gb[AxisNo.Allocate_Y].Admin._OpMode.en := E_AXIS_MODE.ModeVel;
ELSIF AllocateManualCommand.AllocatedRobot.AxisY.JOG.MoveBWD AND AllowAllocateRobotMove THEN
    arAxisCtrl_gb[AxisNo.Allocate_Y].VelMode.Acc := CurrentData.Axes.Allocate_Y.Manual.JogAcceleration;
    arAxisCtrl_gb[AxisNo.Allocate_Y].VelMode.Dec := CurrentData.Axes.Allocate_Y.Manual.JogDeceleration;
    arAxisCtrl_gb[AxisNo.Allocate_Y].VelMode.Jerk := CurrentData.Axes.Allocate_Y.Manual.JogJerk;
    arAxisCtrl_gb[AxisNo.Allocate_Y].VelMode.Velocity := CurrentData.Axes.Allocate_Y.Manual.JogVelocity * -1;
    arAxisCtrl_gb[AxisNo.Allocate_Y].Admin._OpMode.en := E_AXIS_MODE.ModeVel;
ELSIF AllocateManualCommand.AllocatedRobot.AxisY.PTP.Enable  AND AllowAllocateRobotMove THEN
    arAxisCtrl_gb[AxisNo.Allocate_Y].PosMode.Acc := CurrentData.Axes.Allocate_Y.Manual.PtpAcceleration;
    arAxisCtrl_gb[AxisNo.Allocate_Y].PosMode.Dec := CurrentData.Axes.Allocate_Y.Manual.PtpDeceleration;
    arAxisCtrl_gb[AxisNo.Allocate_Y].PosMode.Jerk := CurrentData.Axes.Allocate_Y.Manual.PtpJerk;
    arAxisCtrl_gb[AxisNo.Allocate_Y].PosMode.Velocity := CurrentData.Axes.Allocate_Y.Manual.PtpVelocity;
    arAxisCtrl_gb[AxisNo.Allocate_Y].PosMode.Position := CurrentData.Axes.Allocate_Y.Manual.PtpPosition;
    arAxisCtrl_gb[AxisNo.Allocate_Y].Admin._OpMode.en := ModePosAbs;
//ELSIF( AllocateManualCommand.AllocatedRobot.AxisY.Homing.Execute OR  fbAllocateArea.fbAllocateHome.AxisHomingRequest ) AND AllowAllocateRobotMove THEN
//    arAxisCtrl_gb[AxisNo.Allocate_Y].SetupMode.eHomingMode := E_HomingMode._36_MoveToAbsHomePoint;
//    arAxisCtrl_gb[AxisNo.Allocate_Y].SetupMode.FastVelo := CurrentData.Axes.Allocate_Y.Homing.FastVelo;
//    arAxisCtrl_gb[AxisNo.Allocate_Y].SetupMode.SlowVelo := CurrentData.Axes.Allocate_Y.Homing.SlowVelo;
//    arAxisCtrl_gb[AxisNo.Allocate_Y].SetupMode.lrOffset := CurrentData.Axes.Allocate_Y.Homing.Offset;
//    arAxisCtrl_gb[AxisNo.Allocate_Y].SetupMode.lrSetPosition := CurrentData.Axes.Allocate_Y.Homing.SetAbsolutePosition;
//    arAxisCtrl_gb[AxisNo.Allocate_Y].SetupMode.stPosBiasParameter.bSetPostionBias := FALSE;
//    arAxisCtrl_gb[AxisNo.Allocate_Y].Admin._OpMode.en := ModeHoming;
ELSIF( AllocateManualCommand.AllocatedRobot.AxisY.Homing.Execute OR  fbAllocateArea.fbAllocateHome.AxisHomingRequest ) AND AllowAllocateRobotMove THEN
	GVL_Machine.AllocatYAxisHome := FALSE;
    arAxisCtrl_gb[AxisNo.Allocate_Y].PosMode.Acc := CurrentData.Axes.Allocate_Y.Homing.FastVelo.Acc;
    arAxisCtrl_gb[AxisNo.Allocate_Y].PosMode.Dec := CurrentData.Axes.Allocate_Y.Homing.FastVelo.Dec;
    arAxisCtrl_gb[AxisNo.Allocate_Y].PosMode.Jerk := CurrentData.Axes.Allocate_Y.Homing.FastVelo.Jerk;
    arAxisCtrl_gb[AxisNo.Allocate_Y].PosMode.Velocity := CurrentData.Axes.Allocate_Y.Homing.FastVelo.Velocity;
    arAxisCtrl_gb[AxisNo.Allocate_Y].PosMode.Position := CurrentData.Axes.Allocate_Y.Homing.Offset;
    arAxisCtrl_gb[AxisNo.Allocate_Y].Admin._OpMode.en := ModePosAbs;
		 
    IF arAxisStatus_gb[AxisNo.Allocate_Y].Admin._OpModeAck = ModePosAbs AND arAxisStatus_gb[AxisNo.Allocate_Y].Admin.CmdDone THEN
        GVL_Machine.AllocatYAxisHome := TRUE;
    END_IF
ELSIF TableMove.xBusy AND AllowAllocateRobotMove THEN
    arAxisCtrl_gb[AxisNo.Allocate_Y].Admin._OpMode.en := ModePosAbs;
ELSIF fbAllocateArea.fb_AllocateBatchMode.Busy AND AllowAllocateRobotMove THEN
    arAxisCtrl_gb[AxisNo.Allocate_Y].Admin._OpMode.en := ModePosAbs;
ELSIF fbAllocateArea.fbAllocateRobotNeedlingMove.xBusy AND AllowAllocateRobotMove THEN
	arAxisCtrl_gb[AxisNo.Allocate_Y].PosMode.Acc := CurrentData.Axes.Allocate_Y.Manual.PtpAcceleration;
    arAxisCtrl_gb[AxisNo.Allocate_Y].PosMode.Dec := CurrentData.Axes.Allocate_Y.Manual.PtpDeceleration;
    arAxisCtrl_gb[AxisNo.Allocate_Y].PosMode.Jerk := CurrentData.Axes.Allocate_Y.Manual.PtpJerk;
    arAxisCtrl_gb[AxisNo.Allocate_Y].PosMode.Velocity := CurrentData.Axes.Allocate_Y.Manual.PtpVelocity;
    arAxisCtrl_gb[AxisNo.Allocate_Y].Admin._OpMode.en := ModePosAbs;
ELSE
    arAxisCtrl_gb[AxisNo.Allocate_Y].Admin.StopDeceleration := 1000;
    arAxisCtrl_gb[AxisNo.Allocate_Y].Admin._OpMode.en := E_AXIS_MODE.ModeAH;
END_IF

{EndRegion}

{region "OutRobot AxisX"}
IF AllocateManualCommand.OutRobot.AxisX.JOG.MoveFWD AND AllowOutRobotMove THEN
    arAxisCtrl_gb[AxisNo.OutRobot_X].VelMode.Acc := CurrentData.Axes.OutRobot_X.Manual.JogAcceleration;
    arAxisCtrl_gb[AxisNo.OutRobot_X].VelMode.Dec := CurrentData.Axes.OutRobot_X.Manual.JogDeceleration;
    arAxisCtrl_gb[AxisNo.OutRobot_X].VelMode.Jerk := CurrentData.Axes.OutRobot_X.Manual.JogJerk;
    arAxisCtrl_gb[AxisNo.OutRobot_X].VelMode.Velocity := CurrentData.Axes.OutRobot_X.Manual.JogVelocity;
    arAxisCtrl_gb[AxisNo.OutRobot_X].Admin._OpMode.en := E_AXIS_MODE.ModeVel;
ELSIF AllocateManualCommand.OutRobot.AxisX.JOG.MoveBWD AND AllowOutRobotMove THEN
    arAxisCtrl_gb[AxisNo.OutRobot_X].VelMode.Acc := CurrentData.Axes.OutRobot_X.Manual.JogAcceleration;
    arAxisCtrl_gb[AxisNo.OutRobot_X].VelMode.Dec := CurrentData.Axes.OutRobot_X.Manual.JogDeceleration;
    arAxisCtrl_gb[AxisNo.OutRobot_X].VelMode.Jerk := CurrentData.Axes.OutRobot_X.Manual.JogJerk;
    arAxisCtrl_gb[AxisNo.OutRobot_X].VelMode.Velocity := CurrentData.Axes.OutRobot_X.Manual.JogVelocity * -1;
    arAxisCtrl_gb[AxisNo.OutRobot_X].Admin._OpMode.en := E_AXIS_MODE.ModeVel;
ELSIF AllocateManualCommand.OutRobot.AxisX.PTP.Enable AND AllowOutRobotMove THEN
    arAxisCtrl_gb[AxisNo.OutRobot_X].PosMode.Acc := CurrentData.Axes.OutRobot_X.Manual.PtpAcceleration;
    arAxisCtrl_gb[AxisNo.OutRobot_X].PosMode.Dec := CurrentData.Axes.OutRobot_X.Manual.PtpDeceleration;
    arAxisCtrl_gb[AxisNo.OutRobot_X].PosMode.Jerk := CurrentData.Axes.OutRobot_X.Manual.PtpJerk;
    arAxisCtrl_gb[AxisNo.OutRobot_X].PosMode.Velocity := CurrentData.Axes.OutRobot_X.Manual.PtpVelocity;
    arAxisCtrl_gb[AxisNo.OutRobot_X].PosMode.Position := CurrentData.Axes.OutRobot_X.Manual.PtpPosition;
    arAxisCtrl_gb[AxisNo.OutRobot_X].Admin._OpMode.en := ModePosAbs;
ELSIF (AllocateManualCommand.OutRobot.AxisX.Homing.Execute OR  fbAllocateArea.fbAllocateHome.AxisHomingRequest ) AND AllowOutRobotMove THEN
    arAxisCtrl_gb[AxisNo.OutRobot_X].SetupMode.eHomingMode := E_HomingMode._28_Neg_HomeInnerRight_withLimit;
    arAxisCtrl_gb[AxisNo.OutRobot_X].SetupMode.FastVelo := CurrentData.Axes.OutRobot_X.Homing.FastVelo;
    arAxisCtrl_gb[AxisNo.OutRobot_X].SetupMode.SlowVelo := CurrentData.Axes.OutRobot_X.Homing.SlowVelo;
    arAxisCtrl_gb[AxisNo.OutRobot_X].SetupMode.lrOffset := CurrentData.Axes.OutRobot_X.Homing.Offset;
    arAxisCtrl_gb[AxisNo.OutRobot_X].SetupMode.lrSetPosition := CurrentData.Axes.OutRobot_X.Homing.SetAbsolutePosition;
    arAxisCtrl_gb[AxisNo.OutRobot_X].SetupMode.stPosBiasParameter.bSetPostionBias := TRUE;
    arAxisCtrl_gb[AxisNo.OutRobot_X].Admin._OpMode.en := ModeHoming;
ELSIF TableMove.xBusy AND AllowOutRobotMove THEN
	arAxisCtrl_gb[AxisNo.OutRobot_X].Admin._OpMode.en := ModePosAbs;
ELSIF (AllocateService.AutoMode_BoxMoveReverse.HandShake.Busy 
	  OR AllocateService.AutoMode_EmptyBoxMove.HandShake.Busy 
	  OR AllocateService.AutoMode_RareBoxMove.HandShake.Busy) AND AllowOutRobotMove THEN
	arAxisCtrl_gb[AxisNo.OutRobot_X].PosMode.Acc := CurrentData.Axes.OutRobot_X.HalfAuto.Acceleration;
    arAxisCtrl_gb[AxisNo.OutRobot_X].PosMode.Dec := CurrentData.Axes.OutRobot_X.HalfAuto.Deceleration;
    arAxisCtrl_gb[AxisNo.OutRobot_X].PosMode.Jerk := CurrentData.Axes.OutRobot_X.HalfAuto.Jerk;
    arAxisCtrl_gb[AxisNo.OutRobot_X].PosMode.Velocity := CurrentData.Axes.OutRobot_X.HalfAuto.Velocity;		   
    arAxisCtrl_gb[AxisNo.OutRobot_X].Admin._OpMode.en := ModePosAbs;
ELSE
    arAxisCtrl_gb[AxisNo.OutRobot_X].Admin.StopDeceleration := 1000;
    arAxisCtrl_gb[AxisNo.OutRobot_X].Admin._OpMode.en := E_AXIS_MODE.ModeAH;
END_IF

{Endregion}

{region "OutRobot AxisY"}
IF AllocateManualCommand.OutRobot.AxisY.JOG.MoveFWD AND AllowOutRobotMove THEN
    arAxisCtrl_gb[AxisNo.OutRobot_Y].VelMode.Acc := CurrentData.Axes.OutRobot_Y.Manual.JogAcceleration;
    arAxisCtrl_gb[AxisNo.OutRobot_Y].VelMode.Dec := CurrentData.Axes.OutRobot_Y.Manual.JogDeceleration;
    arAxisCtrl_gb[AxisNo.OutRobot_Y].VelMode.Jerk := CurrentData.Axes.OutRobot_Y.Manual.JogJerk;
    arAxisCtrl_gb[AxisNo.OutRobot_Y].VelMode.Velocity := CurrentData.Axes.OutRobot_Y.Manual.JogVelocity;
    arAxisCtrl_gb[AxisNo.OutRobot_Y].Admin._OpMode.en := E_AXIS_MODE.ModeVel;
ELSIF AllocateManualCommand.OutRobot.AxisY.JOG.MoveBWD AND AllowOutRobotMove THEN
    arAxisCtrl_gb[AxisNo.OutRobot_Y].VelMode.Acc := CurrentData.Axes.OutRobot_Y.Manual.JogAcceleration;
    arAxisCtrl_gb[AxisNo.OutRobot_Y].VelMode.Dec := CurrentData.Axes.OutRobot_Y.Manual.JogDeceleration;
    arAxisCtrl_gb[AxisNo.OutRobot_Y].VelMode.Jerk := CurrentData.Axes.OutRobot_Y.Manual.JogJerk;
    arAxisCtrl_gb[AxisNo.OutRobot_Y].VelMode.Velocity := CurrentData.Axes.OutRobot_Y.Manual.JogVelocity * -1;
    arAxisCtrl_gb[AxisNo.OutRobot_Y].Admin._OpMode.en := E_AXIS_MODE.ModeVel;
ELSIF AllocateManualCommand.OutRobot.AxisY.PTP.Enable AND AllowOutRobotMove THEN
    arAxisCtrl_gb[AxisNo.OutRobot_Y].PosMode.Acc := CurrentData.Axes.OutRobot_Y.Manual.PtpAcceleration;
    arAxisCtrl_gb[AxisNo.OutRobot_Y].PosMode.Dec := CurrentData.Axes.OutRobot_Y.Manual.PtpDeceleration;
    arAxisCtrl_gb[AxisNo.OutRobot_Y].PosMode.Jerk := CurrentData.Axes.OutRobot_Y.Manual.PtpJerk;
    arAxisCtrl_gb[AxisNo.OutRobot_Y].PosMode.Velocity := CurrentData.Axes.OutRobot_Y.Manual.PtpVelocity;
    arAxisCtrl_gb[AxisNo.OutRobot_Y].PosMode.Position := CurrentData.Axes.OutRobot_Y.Manual.PtpPosition;
    arAxisCtrl_gb[AxisNo.OutRobot_Y].Admin._OpMode.en := ModePosAbs;
ELSIF (AllocateManualCommand.OutRobot.AxisY.Homing.Execute OR  fbAllocateArea.fbAllocateHome.AxisHomingRequest) AND AllowOutRobotMove THEN
    arAxisCtrl_gb[AxisNo.OutRobot_Y].SetupMode.eHomingMode := E_HomingMode._28_Neg_HomeInnerRight_withLimit;
    arAxisCtrl_gb[AxisNo.OutRobot_Y].SetupMode.FastVelo := CurrentData.Axes.OutRobot_Y.Homing.FastVelo;
    arAxisCtrl_gb[AxisNo.OutRobot_Y].SetupMode.SlowVelo := CurrentData.Axes.OutRobot_Y.Homing.SlowVelo;
    arAxisCtrl_gb[AxisNo.OutRobot_Y].SetupMode.lrOffset := CurrentData.Axes.OutRobot_Y.Homing.Offset;
    arAxisCtrl_gb[AxisNo.OutRobot_Y].SetupMode.lrSetPosition := CurrentData.Axes.OutRobot_Y.Homing.SetAbsolutePosition;
    arAxisCtrl_gb[AxisNo.OutRobot_Y].SetupMode.stPosBiasParameter.bSetPostionBias := TRUE;
    arAxisCtrl_gb[AxisNo.OutRobot_Y].Admin._OpMode.en := ModeHoming;
ELSIF TableMove.xBusy AND AllowOutRobotMove THEN
	arAxisCtrl_gb[AxisNo.OutRobot_Y].Admin._OpMode.en := ModePosAbs;
ELSIF (AllocateService.AutoMode_BoxMoveReverse.HandShake.Busy 
	  OR AllocateService.AutoMode_EmptyBoxMove.HandShake.Busy 
	  OR AllocateService.AutoMode_RareBoxMove.HandShake.Busy)AND AllowOutRobotMove THEN
	arAxisCtrl_gb[AxisNo.OutRobot_Y].PosMode.Acc := CurrentData.Axes.OutRobot_Y.HalfAuto.Acceleration;
    arAxisCtrl_gb[AxisNo.OutRobot_Y].PosMode.Dec := CurrentData.Axes.OutRobot_Y.HalfAuto.Deceleration;
    arAxisCtrl_gb[AxisNo.OutRobot_Y].PosMode.Jerk := CurrentData.Axes.OutRobot_Y.HalfAuto.Jerk;
    arAxisCtrl_gb[AxisNo.OutRobot_Y].PosMode.Velocity := CurrentData.Axes.OutRobot_Y.HalfAuto.Velocity;		   
    arAxisCtrl_gb[AxisNo.OutRobot_Y].Admin._OpMode.en := ModePosAbs;
ELSE
    arAxisCtrl_gb[AxisNo.OutRobot_Y].Admin.StopDeceleration := 1000;
    arAxisCtrl_gb[AxisNo.OutRobot_Y].Admin._OpMode.en := E_AXIS_MODE.ModeAH;
END_IF

{Endregion}

{region "RoundBelt Axis"}
IF AllocateManualCommand.RoundBelt.Axis.JOG.MoveFWD AND AllowRoundBeltMove THEN
    arAxisCtrl_gb[AxisNo.RoundBelt].VelMode.Acc := CurrentData.Axes.RoundBelt.Manual.JogAcceleration;
    arAxisCtrl_gb[AxisNo.RoundBelt].VelMode.Dec := CurrentData.Axes.RoundBelt.Manual.JogDeceleration;
    arAxisCtrl_gb[AxisNo.RoundBelt].VelMode.Jerk := CurrentData.Axes.RoundBelt.Manual.JogJerk;
    arAxisCtrl_gb[AxisNo.RoundBelt].VelMode.Velocity := CurrentData.Axes.RoundBelt.Manual.JogVelocity;
    arAxisCtrl_gb[AxisNo.RoundBelt].Admin._OpMode.en := E_AXIS_MODE.ModeVel;
ELSIF AllocateManualCommand.RoundBelt.Axis.JOG.MoveBWD AND AllowRoundBeltMove THEN
    arAxisCtrl_gb[AxisNo.RoundBelt].VelMode.Acc := CurrentData.Axes.RoundBelt.Manual.JogAcceleration;
    arAxisCtrl_gb[AxisNo.RoundBelt].VelMode.Dec := CurrentData.Axes.RoundBelt.Manual.JogDeceleration;
    arAxisCtrl_gb[AxisNo.RoundBelt].VelMode.Jerk := CurrentData.Axes.RoundBelt.Manual.JogJerk;
    arAxisCtrl_gb[AxisNo.RoundBelt].VelMode.Velocity := CurrentData.Axes.RoundBelt.Manual.JogVelocity * -1;
    arAxisCtrl_gb[AxisNo.RoundBelt].Admin._OpMode.en := E_AXIS_MODE.ModeVel;
ELSIF AllocateManualCommand.RoundBelt.Axis.PTP.Enable AND AllowRoundBeltMove THEN
    arAxisCtrl_gb[AxisNo.RoundBelt].PosMode.Acc := CurrentData.Axes.RoundBelt.Manual.PtpAcceleration;
    arAxisCtrl_gb[AxisNo.RoundBelt].PosMode.Dec := CurrentData.Axes.RoundBelt.Manual.PtpDeceleration;
    arAxisCtrl_gb[AxisNo.RoundBelt].PosMode.Jerk := CurrentData.Axes.RoundBelt.Manual.PtpJerk;
    arAxisCtrl_gb[AxisNo.RoundBelt].PosMode.Velocity := CurrentData.Axes.RoundBelt.Manual.PtpVelocity;
    arAxisCtrl_gb[AxisNo.RoundBelt].PosMode.Position := CurrentData.Axes.RoundBelt.Manual.PtpPosition;
    arAxisCtrl_gb[AxisNo.RoundBelt].Admin._OpMode.en := ModePosAbs;
ELSIF (AllocateManualCommand.RoundBelt.Axis.Homing.Execute OR  fbAllocateArea.fbAllocateHome.AxisHomingRequest ) AND AllowRoundBeltMove THEN
    arAxisCtrl_gb[AxisNo.RoundBelt].SetupMode.eHomingMode := E_HomingMode._20_Pos_HomeInnerLeft;
    arAxisCtrl_gb[AxisNo.RoundBelt].SetupMode.FastVelo := CurrentData.Axes.RoundBelt.Homing.FastVelo;
    arAxisCtrl_gb[AxisNo.RoundBelt].SetupMode.SlowVelo := CurrentData.Axes.RoundBelt.Homing.SlowVelo;
    arAxisCtrl_gb[AxisNo.RoundBelt].SetupMode.lrOffset := CurrentData.Axes.RoundBelt.Homing.Offset;
    arAxisCtrl_gb[AxisNo.RoundBelt].SetupMode.lrSetPosition := CurrentData.Axes.RoundBelt.Homing.SetAbsolutePosition;
    arAxisCtrl_gb[AxisNo.RoundBelt].SetupMode.stPosBiasParameter.bSetPostionBias := TRUE;
    arAxisCtrl_gb[AxisNo.RoundBelt].Admin._OpMode.en := ModeHoming;
ELSIF TableMove.xBusy AND AllowRoundBeltMove THEN
    arAxisCtrl_gb[AxisNo.RoundBelt].Admin._OpMode.en := ModePosAbs;
ELSIF AllocateService.AllocateCircleMove.HandShake.Busy AND AllowRoundBeltMove THEN
    arAxisCtrl_gb[AxisNo.RoundBelt].PosMode.Acc := CurrentData.Axes.RoundBelt.HalfAuto.Acceleration;
    arAxisCtrl_gb[AxisNo.RoundBelt].PosMode.Dec := CurrentData.Axes.RoundBelt.HalfAuto.Deceleration;
    arAxisCtrl_gb[AxisNo.RoundBelt].PosMode.Jerk := CurrentData.Axes.RoundBelt.HalfAuto.Jerk;
    arAxisCtrl_gb[AxisNo.RoundBelt].PosMode.Velocity := CurrentData.Axes.RoundBelt.HalfAuto.Velocity;
    arAxisCtrl_gb[AxisNo.RoundBelt].Admin._OpMode.en := ModePosAbs;
ELSIF (AllocateService.AutoMode_AllocateBatchMode.HandShake.Busy OR StorageService.AutoMode_ReloadRoundBeltBoxWithRobot.Status.Busy) AND AllowRoundBeltMove THEN
    arAxisCtrl_gb[AxisNo.RoundBelt].PosMode.Acc := CurrentData.Axes.RoundBelt.HalfAuto.Acceleration;
    arAxisCtrl_gb[AxisNo.RoundBelt].PosMode.Dec := CurrentData.Axes.RoundBelt.HalfAuto.Deceleration;
    arAxisCtrl_gb[AxisNo.RoundBelt].PosMode.Jerk := CurrentData.Axes.RoundBelt.HalfAuto.Jerk;
    arAxisCtrl_gb[AxisNo.RoundBelt].PosMode.Velocity := CurrentData.Axes.RoundBelt.HalfAuto.Velocity;
    arAxisCtrl_gb[AxisNo.RoundBelt].Admin._OpMode.en := ModePosAbs;
ELSE
    arAxisCtrl_gb[AxisNo.RoundBelt].Admin.StopDeceleration := 1000;
    arAxisCtrl_gb[AxisNo.RoundBelt].Admin._OpMode.en := E_AXIS_MODE.ModeAH;
END_IF

{endregion}

{region "TurnTable Axis"}
IF AllocateManualCommand.TurnTable.Axis.JOG.MoveFWD AND AllowTurnTable THEN
    arAxisCtrl_gb[AxisNo.TurnTable].VelMode.Acc := CurrentData.Axes.TurnTable.Manual.JogAcceleration;
    arAxisCtrl_gb[AxisNo.TurnTable].VelMode.Dec := CurrentData.Axes.TurnTable.Manual.JogDeceleration;
    arAxisCtrl_gb[AxisNo.TurnTable].VelMode.Jerk := CurrentData.Axes.TurnTable.Manual.JogJerk;
    arAxisCtrl_gb[AxisNo.TurnTable].VelMode.Velocity := CurrentData.Axes.TurnTable.Manual.JogVelocity;
    arAxisCtrl_gb[AxisNo.TurnTable].Admin._OpMode.en := E_AXIS_MODE.ModeVel;
ELSIF AllocateManualCommand.TurnTable.Axis.JOG.MoveBWD THEN
    arAxisCtrl_gb[AxisNo.TurnTable].VelMode.Acc := CurrentData.Axes.TurnTable.Manual.JogAcceleration;
    arAxisCtrl_gb[AxisNo.TurnTable].VelMode.Dec := CurrentData.Axes.TurnTable.Manual.JogDeceleration;
    arAxisCtrl_gb[AxisNo.TurnTable].VelMode.Jerk := CurrentData.Axes.TurnTable.Manual.JogJerk;
    arAxisCtrl_gb[AxisNo.TurnTable].VelMode.Velocity := CurrentData.Axes.TurnTable.Manual.JogVelocity * -1;
    arAxisCtrl_gb[AxisNo.TurnTable].Admin._OpMode.en := E_AXIS_MODE.ModeVel;
ELSIF AllocateManualCommand.TurnTable.Axis.PTP.Enable THEN
    arAxisCtrl_gb[AxisNo.TurnTable].PosMode.Acc := CurrentData.Axes.TurnTable.Manual.PtpAcceleration;
    arAxisCtrl_gb[AxisNo.TurnTable].PosMode.Dec := CurrentData.Axes.TurnTable.Manual.PtpDeceleration;
    arAxisCtrl_gb[AxisNo.TurnTable].PosMode.Jerk := CurrentData.Axes.TurnTable.Manual.PtpJerk;
    arAxisCtrl_gb[AxisNo.TurnTable].PosMode.Velocity := CurrentData.Axes.TurnTable.Manual.PtpVelocity;
    arAxisCtrl_gb[AxisNo.TurnTable].PosMode.Position := CurrentData.Axes.TurnTable.Manual.PtpPosition;
    arAxisCtrl_gb[AxisNo.TurnTable].Admin._OpMode.en := ModePosAbs;
ELSIF (AllocateManualCommand.TurnTable.Axis.Homing.Execute OR  fbAllocateArea.fbAllocateHome.AxisHomingRequest) AND  AllowTurnTable THEN
    arAxisCtrl_gb[AxisNo.TurnTable].SetupMode.eHomingMode := E_HomingMode._22_Neg_HomeInnerRight;
    arAxisCtrl_gb[AxisNo.TurnTable].SetupMode.FastVelo := CurrentData.Axes.TurnTable.Homing.FastVelo;
    arAxisCtrl_gb[AxisNo.TurnTable].SetupMode.SlowVelo := CurrentData.Axes.TurnTable.Homing.SlowVelo;
    arAxisCtrl_gb[AxisNo.TurnTable].SetupMode.lrOffset := CurrentData.Axes.TurnTable.Homing.Offset;
    arAxisCtrl_gb[AxisNo.TurnTable].SetupMode.lrSetPosition := CurrentData.Axes.TurnTable.Homing.SetAbsolutePosition;
    arAxisCtrl_gb[AxisNo.TurnTable].SetupMode.stPosBiasParameter.bSetPostionBias := TRUE;
    arAxisCtrl_gb[AxisNo.TurnTable].Admin._OpMode.en := ModeHoming;
ELSIF TableMove.xBusy AND AllowTurnTable THEN
    arAxisCtrl_gb[AxisNo.TurnTable].Admin._OpMode.en := ModePosAbs;
ELSIF AllocateService.TurnTableMove.HandShake.Busy AND fbAllocateArea.TurnTableControl.bTurnTableMoveRequest AND AllowTurnTable THEN
    arAxisCtrl_gb[AxisNo.TurnTable].PosMode.Acc := CurrentData.Axes.TurnTable.HalfAuto.Acceleration;
    arAxisCtrl_gb[AxisNo.TurnTable].PosMode.Dec := CurrentData.Axes.TurnTable.HalfAuto.Deceleration;
    arAxisCtrl_gb[AxisNo.TurnTable].PosMode.Jerk := CurrentData.Axes.TurnTable.HalfAuto.Jerk;
    arAxisCtrl_gb[AxisNo.TurnTable].PosMode.Velocity := CurrentData.Axes.TurnTable.HalfAuto.Velocity;
    arAxisCtrl_gb[AxisNo.TurnTable].Admin._OpMode.en := ModePosAbs;
ELSE
    arAxisCtrl_gb[AxisNo.TurnTable].Admin.StopDeceleration := 1000;
    arAxisCtrl_gb[AxisNo.TurnTable].Admin._OpMode.en := E_AXIS_MODE.ModeAH;
END_IF

{endregion}

IF NOT (fbStorageArea.RackState = E_RackState.FeedBox) AND 
	NOT (fbStorageArea.RackState = E_RackState.TransitingFeedBox) OR 
	fbStorageArea.fbStorageHoming.xBusy THEN
			
		IF StorageManualCommand.RackMotor.Axis.JOG.MoveFWD AND AllowRackMotor THEN
			arAxisCtrl_gb[AxisNo.RackMotor].VelMode.Acc := CurrentData.Axes.RackMotor.Manual.JogAcceleration;
			arAxisCtrl_gb[AxisNo.RackMotor].VelMode.Dec := CurrentData.Axes.RackMotor.Manual.JogDeceleration;
			arAxisCtrl_gb[AxisNo.RackMotor].VelMode.Jerk := CurrentData.Axes.RackMotor.Manual.JogJerk;
			arAxisCtrl_gb[AxisNo.RackMotor].VelMode.Velocity := CurrentData.Axes.RackMotor.Manual.JogVelocity;
			arAxisCtrl_gb[AxisNo.RackMotor].Admin._OpMode.en := E_AXIS_MODE.ModeVel;
		ELSIF StorageManualCommand.RackMotor.Axis.JOG.MoveBWD AND AllowRackMotor THEN
			arAxisCtrl_gb[AxisNo.RackMotor].VelMode.Acc := CurrentData.Axes.RackMotor.Manual.JogAcceleration;
			arAxisCtrl_gb[AxisNo.RackMotor].VelMode.Dec := CurrentData.Axes.RackMotor.Manual.JogDeceleration;
			arAxisCtrl_gb[AxisNo.RackMotor].VelMode.Jerk := CurrentData.Axes.RackMotor.Manual.JogJerk;
			arAxisCtrl_gb[AxisNo.RackMotor].VelMode.Velocity := CurrentData.Axes.RackMotor.Manual.JogVelocity * -1;
			arAxisCtrl_gb[AxisNo.RackMotor].Admin._OpMode.en := E_AXIS_MODE.ModeVel;
		ELSIF StorageManualCommand.RackMotor.Axis.PTP.Enable AND AllowRackMotor THEN
			arAxisCtrl_gb[AxisNo.RackMotor].PosMode.Acc := CurrentData.Axes.RackMotor.Manual.PtpAcceleration;
			arAxisCtrl_gb[AxisNo.RackMotor].PosMode.Dec := CurrentData.Axes.RackMotor.Manual.PtpDeceleration;
			arAxisCtrl_gb[AxisNo.RackMotor].PosMode.Jerk := CurrentData.Axes.RackMotor.Manual.PtpJerk;
			arAxisCtrl_gb[AxisNo.RackMotor].PosMode.Velocity := CurrentData.Axes.RackMotor.Manual.PtpVelocity;
			arAxisCtrl_gb[AxisNo.RackMotor].PosMode.Position := CurrentData.Axes.RackMotor.Manual.PtpPosition;
			arAxisCtrl_gb[AxisNo.RackMotor].Admin._OpMode.en := ModePosAbs;
		ELSIF (StorageManualCommand.RackMotor.Axis.Homing.Execute OR fbStorageArea.fbStorageHoming.RackMotorHomeRequest) AND AllowRackMotor THEN
			arAxisCtrl_gb[AxisNo.RackMotor].SetupMode.eHomingMode := E_HomingMode._17_Neg_LimitOutterRight;
			arAxisCtrl_gb[AxisNo.RackMotor].SetupMode.FastVelo := CurrentData.Axes.RackMotor.Homing.FastVelo;
			arAxisCtrl_gb[AxisNo.RackMotor].SetupMode.SlowVelo := CurrentData.Axes.RackMotor.Homing.SlowVelo;
			arAxisCtrl_gb[AxisNo.RackMotor].SetupMode.lrOffset := CurrentData.Axes.RackMotor.Homing.Offset;
			arAxisCtrl_gb[AxisNo.RackMotor].SetupMode.lrSetPosition := CurrentData.Axes.RackMotor.Homing.SetAbsolutePosition;
			arAxisCtrl_gb[AxisNo.RackMotor].SetupMode.stPosBiasParameter.bSetPostionBias := TRUE;
			arAxisCtrl_gb[AxisNo.RackMotor].Admin._OpMode.en := ModeHoming;
		ELSIF (TableMove.xBusy OR StorageService.AutoMode_AddBoxes.Status.Busy) AND AllowRackMotor THEN
			arAxisCtrl_gb[AxisNo.RackMotor].Admin._OpMode.en := ModePosAbs;
		ELSE
			arAxisCtrl_gb[AxisNo.RackMotor].Admin.StopDeceleration := 1000;
			arAxisCtrl_gb[AxisNo.RackMotor].Admin._OpMode.en := E_AXIS_MODE.ModeAH;
		END_IF
ELSIF fbStorageArea.fbBoxSupplyCtrl.Busy AND 
			fbStorageArea.fbBoxSupplyCtrl.AxisRackMotorBTNHomeRequest AND 
			AllowRackMotor THEN
		arAxisCtrl_gb[AxisNo.RackMotor].PosMode.Acc := CurrentData.Axes.RackMotor.HalfAuto.Acceleration;
		arAxisCtrl_gb[AxisNo.RackMotor].PosMode.Dec := CurrentData.Axes.RackMotor.HalfAuto.Deceleration;
		arAxisCtrl_gb[AxisNo.RackMotor].PosMode.Jerk := CurrentData.Axes.RackMotor.HalfAuto.Jerk;
		arAxisCtrl_gb[AxisNo.RackMotor].PosMode.Velocity := CurrentData.Axes.RackMotor.HalfAuto.Velocity;
		arAxisCtrl_gb[AxisNo.RackMotor].Admin._OpMode.en := ModePosAbs;	  
ELSE
		arAxisCtrl_gb[AxisNo.RackMotor].Admin.StopDeceleration := 1000;
		arAxisCtrl_gb[AxisNo.RackMotor].Admin._OpMode.en := E_AXIS_MODE.ModeAH;	 
END_IF
END_METHOD

METHOD PRIVATE M_Manual_Cylinder
VAR_INPUT
END_VAR
CylinderManualCtrl[1](bTrigger 	:=StorageManualCommand.UpCV.FeedInPress1.Exetend);
CylinderManualCtrl[2](bTrigger 	:=StorageManualCommand.UpCV.FeedInPress2.Exetend);
CylinderManualCtrl[3](bTrigger 	:=StorageManualCommand.UpCV.DiameterPress.Exetend);
CylinderManualCtrl[4](bTrigger 	:=StorageManualCommand.UpCV.CamaraPress1.Exetend);
CylinderManualCtrl[5](bTrigger 	:=StorageManualCommand.UpCV.CamaraPress2.Exetend);
CylinderManualCtrl[6](bTrigger 	:=StorageManualCommand.UpCV.CamaraPress3.Exetend);
CylinderManualCtrl[7](bTrigger 	:=StorageManualCommand.UpCV.CamaraPress4.Exetend);
CylinderManualCtrl[8](bTrigger 	:=StorageManualCommand.UpCV.Block1.Exetend);
CylinderManualCtrl[9](bTrigger 	:=StorageManualCommand.UpCV.Block2.Exetend);
CylinderManualCtrl[10](bTrigger :=StorageManualCommand.UpCV.Block3.Exetend);
CylinderManualCtrl[11](bTrigger :=StorageManualCommand.UpCV.DiameterHoriz.Exetend,
					   Hold 	:= NOT Cylinder.List.fbUpCV_DiameterVert.InRearPosition);
CylinderManualCtrl[12](bTrigger	:=StorageManualCommand.UpCV.DiameterVert.Exetend);
CylinderManualCtrl[13](bTrigger	:=StorageManualCommand.UpCV.DiameterClamp.Exetend);
CylinderManualCtrl[14](bTrigger	:=StorageManualCommand.UpCV.StackPush.Exetend,
						Hold	:= NOT arAxisCtrl_gb[AxisNo.RackMotor].Admin.Axis.Status.NotMoving);
CylinderManualCtrl[15](bTrigger	:=AllocateManualCommand.PullOutCV.AsidePress1.Exetend);
CylinderManualCtrl[16](bTrigger	:=AllocateManualCommand.PullOutCV.AsidePress2.Exetend);
CylinderManualCtrl[17](bTrigger	:=AllocateManualCommand.PullOutCV.AsideBlock.Exetend);
CylinderManualCtrl[18](bTrigger	:=AllocateManualCommand.PullOutCV.BsidePress1.Exetend);
CylinderManualCtrl[19](bTrigger	:=AllocateManualCommand.PullOutCV.BsidePress2.Exetend);
CylinderManualCtrl[20](bTrigger	:=AllocateManualCommand. PullOutCV.BsideBlock.Exetend);
CylinderManualCtrl[21](bTrigger	:=StorageManualCommand.LowCV.Press1.Exetend);
CylinderManualCtrl[22](bTrigger	:=StorageManualCommand.LowCV.Press2.Exetend);
CylinderManualCtrl[23](bTrigger	:=StorageManualCommand.LowCV.Press3.Exetend);
CylinderManualCtrl[24](bTrigger	:=StorageManualCommand.LowCV.Press4.Exetend);
CylinderManualCtrl[25](bTrigger	:=StorageManualCommand.LowCV.Block1.Exetend);
CylinderManualCtrl[26](bTrigger	:=StorageManualCommand.LowCV.Block2.Exetend);
CylinderManualCtrl[27](bTrigger	:=AllocateManualCommand.AllocatedRobot.LeftVert1.Exetend,
						Hold	:= 	(NOT arAxisCtrl_gb[AxisNo.RoundBelt].Admin.Axis.Status.NotMoving)
								OR  (NOT arAxisCtrl_gb[AxisNo.TurnTable].Admin.Axis.Status.NotMoving)
								OR  (NOT arAxisCtrl_gb[AxisNo.Allocate_X].Admin.Axis.Status.NotMoving)
								OR  (NOT arAxisCtrl_gb[AxisNo.Allocate_Y].Admin.Axis.Status.NotMoving));
CylinderManualCtrl[28](bTrigger	:=AllocateManualCommand.AllocatedRobot.LeftVert2.Exetend,
						Hold	:= 	(NOT arAxisCtrl_gb[AxisNo.RoundBelt].Admin.Axis.Status.NotMoving)
								OR  (NOT arAxisCtrl_gb[AxisNo.TurnTable].Admin.Axis.Status.NotMoving)
								OR  (NOT arAxisCtrl_gb[AxisNo.Allocate_X].Admin.Axis.Status.NotMoving)
								OR  (NOT arAxisCtrl_gb[AxisNo.Allocate_Y].Admin.Axis.Status.NotMoving));

CylinderManualCtrl[29](bTrigger	:=AllocateManualCommand.AllocatedRobot.RightVert1.Exetend,
						Hold	:= 	(NOT arAxisCtrl_gb[AxisNo.RoundBelt].Admin.Axis.Status.NotMoving)
								OR  (NOT arAxisCtrl_gb[AxisNo.TurnTable].Admin.Axis.Status.NotMoving)
								OR  (NOT arAxisCtrl_gb[AxisNo.Allocate_X].Admin.Axis.Status.NotMoving)
								OR  (NOT arAxisCtrl_gb[AxisNo.Allocate_Y].Admin.Axis.Status.NotMoving));

CylinderManualCtrl[30](bTrigger	:=AllocateManualCommand.AllocatedRobot.RightVert2.Exetend,
						Hold	:= 	(NOT arAxisCtrl_gb[AxisNo.RoundBelt].Admin.Axis.Status.NotMoving)
								OR  (NOT arAxisCtrl_gb[AxisNo.TurnTable].Admin.Axis.Status.NotMoving)
								OR  (NOT arAxisCtrl_gb[AxisNo.Allocate_X].Admin.Axis.Status.NotMoving)
								OR  (NOT arAxisCtrl_gb[AxisNo.Allocate_Y].Admin.Axis.Status.NotMoving));
CylinderManualCtrl[31](bTrigger	:=AllocateManualCommand.AllocatedRobot.LeftClamp1.Exetend);
CylinderManualCtrl[32](bTrigger	:=AllocateManualCommand.AllocatedRobot.LeftClamp2.Exetend);
CylinderManualCtrl[33](bTrigger	:=AllocateManualCommand.AllocatedRobot.RightClamp1.Exetend);
CylinderManualCtrl[34](bTrigger	:=AllocateManualCommand.AllocatedRobot.RightClamp2.Exetend);
CylinderManualCtrl[35](bTrigger	:=AllocateManualCommand.RoundBelt.WorkZone_Press.Exetend,
						Hold	:= NOT arAxisCtrl_gb[AxisNo.RoundBelt].Admin.Axis.Status.NotMoving);
CylinderManualCtrl[36](bTrigger	:=AllocateManualCommand.RoundBelt.WorkZone_Plug.Exetend,
						Hold	:= NOT arAxisCtrl_gb[AxisNo.RoundBelt].Admin.Axis.Status.NotMoving);
CylinderManualCtrl[37](bTrigger	:=AllocateManualCommand.RoundBelt.ChargeZone_Plug.Exetend,
						Hold	:= NOT arAxisCtrl_gb[AxisNo.RoundBelt].Admin.Axis.Status.NotMoving);
						
CylinderManualCtrl[38](bTrigger	:=AllocateManualCommand.RoundBelt.TransmitCVZone_Plug.Exetend,
						Hold	:= NOT arAxisCtrl_gb[AxisNo.RoundBelt].Admin.Axis.Status.NotMoving);
						
CylinderManualCtrl[39](bTrigger	:=AllocateManualCommand.OutRobot.AsideVert.Exetend,
						Hold	:= (NOT arAxisCtrl_gb[AxisNo.TurnTable].Admin.Axis.Status.NotMoving) 
								OR (NOT  arAxisCtrl_gb[AxisNo.OutRobot_X].Admin.Axis.Status.NotMoving)
								OR (NOT  arAxisCtrl_gb[AxisNo.OutRobot_Y].Admin.Axis.Status.NotMoving));
						
CylinderManualCtrl[40](bTrigger	:=AllocateManualCommand.OutRobot.BsideVert.Exetend,
						Hold	:= (NOT arAxisCtrl_gb[AxisNo.TurnTable].Admin.Axis.Status.NotMoving)
								OR (NOT  arAxisCtrl_gb[AxisNo.OutRobot_X].Admin.Axis.Status.NotMoving) 
								OR (NOT  arAxisCtrl_gb[AxisNo.OutRobot_Y].Admin.Axis.Status.NotMoving));
CylinderManualCtrl[41](bTrigger	:=AllocateManualCommand.OutRobot.AsideClamp.Exetend);
CylinderManualCtrl[42](bTrigger	:=AllocateManualCommand.OutRobot.BsideClamp.Exetend);
CylinderManualCtrl[43](bTrigger	:=AllocateManualCommand.TransCV.CamaraHoriz .Exetend);
CylinderManualCtrl[44](bTrigger	:=AllocateManualCommand.TransCV.DifferentSizeCV_Press2.Exetend);
CylinderManualCtrl[45](bTrigger	:=AllocateManualCommand.TransCV.DifferentSizeCV_Press1.Exetend);
CylinderManualCtrl[46](bTrigger	:=AllocateManualCommand.TransCV.DifferentSizeCV_Block1.Exetend);
CylinderManualCtrl[47](bTrigger	:=AllocateManualCommand.TransCV.SameSizeCV_Press4.Exetend);
CylinderManualCtrl[48](bTrigger	:=AllocateManualCommand.TransCV.SameSizeCV_Press3.Exetend);
CylinderManualCtrl[49](bTrigger	:=AllocateManualCommand.TransCV.SameSizeCV_Press2.Exetend);
CylinderManualCtrl[50](bTrigger	:=AllocateManualCommand.TransCV.SameSizeCV_Press1.Exetend);
CylinderManualCtrl[51](bTrigger	:=AllocateManualCommand.TransCV.SameSizeCV_Block2.Exetend);
CylinderManualCtrl[52](bTrigger	:=AllocateManualCommand.TransCV.SameSizeCV_Block1 .Exetend);
CylinderManualCtrl[53](bTrigger	:=AllocateManualCommand.TurnTable.Press.Exetend,
						Hold	:= NOT arAxisCtrl_gb[AxisNo.TurnTable].Admin.Axis.Status.NotMoving);
END_METHOD

METHOD PRIVATE M_Manual_Motor
VAR_INPUT
END_VAR

MotorManualCtrl[1](bForward  := StorageManualCommand.WareHouseCV_01.Forward,
                   bBackward := StorageManualCommand.WareHouseCV_01.Backward,
                   bStop     := StorageManualCommand.WareHouseCV_01.Stopped,
                   Motor     := Motor.List.WareHouseCV_01);

MotorManualCtrl[2](bForward  := StorageManualCommand.WareHouseCV_02.Forward,
                   bBackward := StorageManualCommand.WareHouseCV_02.Backward,
                   bStop     := StorageManualCommand.WareHouseCV_02.Stopped,
                   Motor     := Motor.List.WareHouseCV_02);

MotorManualCtrl[3](bForward  := StorageManualCommand.WareHouseCV_03.Forward,
                   bBackward := StorageManualCommand.WareHouseCV_03.Backward,
                   bStop     := StorageManualCommand.WareHouseCV_03.Stopped,
                   Motor     := Motor.List.WareHouseCV_03);

MotorManualCtrl[4](bForward  := StorageManualCommand.WareHouseCV_04.Forward,
                   bBackward := StorageManualCommand.WareHouseCV_04.Backward,
                   bStop     := StorageManualCommand.WareHouseCV_04.Stopped,
                   Motor     := Motor.List.WareHouseCV_04);

MotorManualCtrl[5](bForward  := StorageManualCommand.WareHouseCV_05.Forward,
                   bBackward := StorageManualCommand.WareHouseCV_05.Backward,
                   bStop     := StorageManualCommand.WareHouseCV_05.Stopped,
                   Motor     := Motor.List.WareHouseCV_05);

MotorManualCtrl[6](bForward  := StorageManualCommand.WareHouseCV_06.Forward,
                   bBackward := StorageManualCommand.WareHouseCV_06.Backward,
                   bStop     := StorageManualCommand.WareHouseCV_06.Stopped,
                   Motor     := Motor.List.WareHouseCV_06);

MotorManualCtrl[7](bForward  := StorageManualCommand.WareHouseCV_07.Forward,
                   bBackward := StorageManualCommand.WareHouseCV_07.Backward,
                   bStop     := StorageManualCommand.WareHouseCV_07.Stopped,
                   Motor     := Motor.List.WareHouseCV_07);

MotorManualCtrl[8](bForward  := StorageManualCommand.WareHouseCV_08.Forward,
                   bBackward := StorageManualCommand.WareHouseCV_08.Backward,
                   bStop     := StorageManualCommand.WareHouseCV_08.Stopped,
                   Motor     := Motor.List.WareHouseCV_08);

MotorManualCtrl[9](bForward  := StorageManualCommand.WareHouseCV_09.Forward,
                   bBackward := StorageManualCommand.WareHouseCV_09.Backward,
                   bStop     := StorageManualCommand.WareHouseCV_09.Stopped,
                   Motor     := Motor.List.WareHouseCV_09);

MotorManualCtrl[10](bForward  := StorageManualCommand.WareHouseCV_10.Forward,
                    bBackward := StorageManualCommand.WareHouseCV_10.Backward,
                    bStop     := StorageManualCommand.WareHouseCV_10.Stopped,
                    Motor     := Motor.List.WareHouseCV_10);

MotorManualCtrl[11](bForward  := StorageManualCommand.WareHouseCV_11.Forward,
                    bBackward := StorageManualCommand.WareHouseCV_11.Backward,
                    bStop     := StorageManualCommand.WareHouseCV_11.Stopped,
                    Motor     := Motor.List.WareHouseCV_11);

MotorManualCtrl[12](bForward  := StorageManualCommand.WareHouseCV_12.Forward,
                    bBackward := StorageManualCommand.WareHouseCV_12.Backward,
                    bStop     := StorageManualCommand.WareHouseCV_12.Stopped,
                    Motor     := Motor.List.WareHouseCV_12);

MotorManualCtrl[13](bForward  := StorageManualCommand.WareHouseCV_13.Forward,
                    bBackward := StorageManualCommand.WareHouseCV_13.Backward,
                    bStop     := StorageManualCommand.WareHouseCV_13.Stopped,
                    Motor     := Motor.List.WareHouseCV_13);

MotorManualCtrl[14](bForward  := StorageManualCommand.WareHouseCV_14.Forward,
                    bBackward := StorageManualCommand.WareHouseCV_14.Backward,
                    bStop     := StorageManualCommand.WareHouseCV_14.Stopped,
                    Motor     := Motor.List.WareHouseCV_14);

MotorManualCtrl[15](bForward  := StorageManualCommand.WareHouseCV_15.Forward,
                    bBackward := StorageManualCommand.WareHouseCV_15.Backward,
                    bStop     := StorageManualCommand.WareHouseCV_15.Stopped,
                    Motor     := Motor.List.WareHouseCV_15);

MotorManualCtrl[16](bForward  := StorageManualCommand.WareHouseCV_16.Forward,
                    bBackward := StorageManualCommand.WareHouseCV_16.Backward,
                    bStop     := StorageManualCommand.WareHouseCV_16.Stopped,
                    Motor     := Motor.List.WareHouseCV_16);

MotorManualCtrl[17](bForward  := StorageManualCommand.WareHouseCV_17.Forward,
                    bBackward := StorageManualCommand.WareHouseCV_17.Backward,
                    bStop     := StorageManualCommand.WareHouseCV_17.Stopped,
                    Motor     := Motor.List.WareHouseCV_17);

MotorManualCtrl[18](bForward  := StorageManualCommand.WareHouseCV_18.Forward,
                    bBackward := StorageManualCommand.WareHouseCV_18.Backward,
                    bStop     := StorageManualCommand.WareHouseCV_18.Stopped,
                    Motor     := Motor.List.WareHouseCV_18);

MotorManualCtrl[19](bForward  := StorageManualCommand.WareHouseCV_19.Forward,
                    bBackward := StorageManualCommand.WareHouseCV_19.Backward,
                    bStop     := StorageManualCommand.WareHouseCV_19.Stopped,
                    Motor     := Motor.List.WareHouseCV_19);

MotorManualCtrl[20](bForward  := StorageManualCommand.WareHouseCV_20.Forward,
                    bBackward := StorageManualCommand.WareHouseCV_20.Backward,
                    bStop     := StorageManualCommand.WareHouseCV_20.Stopped,
                    Motor     := Motor.List.WareHouseCV_20);

MotorManualCtrl[21](bForward  := StorageManualCommand.UpCV.UpCV.Forward,
                    bBackward := StorageManualCommand.UpCV.UpCV.Backward,
                    bStop     := StorageManualCommand.UpCV.UpCV.Stopped,
					Hold	  := INPUT.bUpCV_DiameterHoriz_RearSensor AND INPUT.bUpCV_DiameterVert_FrontSensor,
                    Motor     := Motor.List.UpCV);

MotorManualCtrl[22](bForward  := StorageManualCommand.LowCV.LowCV.Forward,
                    bBackward := StorageManualCommand.LowCV.LowCV.Backward,
                    bStop     := StorageManualCommand.LowCV.LowCV.Stopped,
                    Motor     := Motor.List.LowCV);

MotorManualCtrl[23](bForward  := AllocateManualCommand.PullOutCV.PullOutCV_A.Forward,
                    bBackward := AllocateManualCommand.PullOutCV.PullOutCV_A.Backward,
                    bStop     := AllocateManualCommand.PullOutCV.PullOutCV_A.Stopped,
                    Motor     := Motor.List.PullOutCV_A);

MotorManualCtrl[24](bForward  := AllocateManualCommand.PullOutCV.PullOutCV_B.Forward,
                    bBackward := AllocateManualCommand.PullOutCV.PullOutCV_B.Backward,
                    bStop     := AllocateManualCommand.PullOutCV.PullOutCV_B.Stopped,
                    Motor     := Motor.List.PullOutCV_B);

MotorManualCtrl[25](bForward  := AllocateManualCommand.TransCV.TransmitSameSideCV.Forward,
                    bBackward := AllocateManualCommand.TransCV.TransmitSameSideCV.Backward,
                    bStop     := AllocateManualCommand.TransCV.TransmitSameSideCV.Stopped,
                    Motor     := Motor.List.TransmitSameSideCV);

MotorManualCtrl[26](bForward  := AllocateManualCommand.TransCV.TransmitDifferentSideCV.Forward,
                    bBackward := AllocateManualCommand.TransCV.TransmitDifferentSideCV.Backward,
                    bStop     := AllocateManualCommand.TransCV.TransmitDifferentSideCV.Stopped,
                    Motor     := Motor.List.TransmitDifferentSideCV);
END_METHOD

METHOD M_ManualAllocateHoming
VAR_INPUT
END_VAR
//fbAllocateArea.fbAllocateHome.xExecute := Service_Handshake.AllocationRegionHome.HandShake.Execute;
IF Service_Handshake.AllocationRegionHome.HandShake.Execute THEN
	fbAllocateArea.M_StartHoming();
END_IF
Service_Handshake.AllocationRegionHome.HandShake.Busy := fbAllocateArea.fbAllocateHome.xBusy;
Service_Handshake.AllocationRegionHome.HandShake.Done := fbAllocateArea.fbAllocateHome.xDone;
Service_Handshake.AllocationRegionHome.HandShake.Error := fbAllocateArea.fbAllocateHome.xError;
IF  NOT Service_Handshake.AllocationRegionHome.HandShake.Execute THEN
	fbAllocateArea.M_StopHoming();
END_IF

Service_Handshake.AllocationRegionHome.Homed := fbAllocateArea.Homed;
END_METHOD

METHOD PRIVATE M_ManualMachineHome
VAR_INPUT
END_VAR
IF Service_Handshake.MachineHome.HandShake.Execute THEN
	M_StartHoming();
END_IF
Service_Handshake.MachineHome.HandShake.Busy := fbMachineHoming.xBusy;
Service_Handshake.MachineHome.HandShake.Done  := fbMachineHoming.xDone;
Service_Handshake.MachineHome.HandShake.Error := fbMachineHoming.xError;
IF NOT Service_Handshake.MachineHome.HandShake.Execute THEN
	M_StopHoming();
END_IF

Service_Handshake.MachineHome.Homed := MachineHomed;
END_METHOD

METHOD M_ManualShippingHoming 
VAR_INPUT
END_VAR
//fbStorageArea.fbStoragehoming.xExecute := Service_Handshake.StorageRegionHome.HandShake.Execute;
IF Service_Handshake.FGARegionHome.HandShake.Execute THEN
	fbShippingArea.M_StartHoming();
END_IF
Service_Handshake.FGARegionHome.HandShake.Busy := fbShippingArea.fbshippinghoming.xBusy;
Service_Handshake.FGARegionHome.HandShake.Done := fbShippingArea.fbshippinghoming.xDone;
Service_Handshake.FGARegionHome.HandShake.Error := fbShippingArea.fbshippinghoming.xError;
IF NOT Service_Handshake.FGARegionHome.HandShake.Execute  THEN
	fbShippingArea.M_StopHoming();
END_IF

Service_Handshake.FGARegionHome.Homed := fbShippingArea.Homed;
END_METHOD

METHOD M_ManualStorageHoming
VAR_INPUT
END_VAR
//fbStorageArea.fbStoragehoming.xExecute := Service_Handshake.StorageRegionHome.HandShake.Execute;
IF Service_Handshake.StorageRegionHome.HandShake.Execute THEN
	fbStorageArea.M_StartHoming();
END_IF
Service_Handshake.StorageRegionHome.HandShake.Busy := fbStorageArea.fbStoragehoming.xBusy;
Service_Handshake.StorageRegionHome.HandShake.Done := fbStorageArea.fbStoragehoming.xDone;
Service_Handshake.StorageRegionHome.HandShake.Error := fbStorageArea.fbStoragehoming.xError;
IF  NOT Service_Handshake.StorageRegionHome.HandShake.Execute THEN
	fbStorageArea.M_StopHoming();
END_IF

Service_Handshake.StorageRegionHome.Homed := fbStorageArea.Homed;
END_METHOD

METHOD M_Resetting
VAR
	CylinderIndex : UDINT;
	MotorIndex : INT;
END_VAR
FOR CylinderIndex := 1 TO udiMax_CylinderNum DO
	fbAllocateArea.M_TransCVCameraPress_ManualMode();
    //Cylinder.arCylinder[CylinderIndex].xEnable := TRUE;
	CylinderManualCtrl[CylinderIndex].Cylinder REF= Cylinder.arCylinder[CylinderIndex];
END_FOR

FOR CylinderIndex := 1 TO udiMax_CylinderNum DO
    Cylinder.arCylinder[CylinderIndex].EnableSimulation := EnableSimulation;
END_FOR

FOR MotorIndex := 1 TO 26 DO
    //Motor.arMotor[MotorIndex].xEnable := TRUE;
	MotorManualCtrl[MotorIndex].Motor REF= Motor.arMotor[MotorIndex];
END_FOR

// Reference 
ReferenceHMI();
RefStorageService();
RefAllocateService();
RefShippingService();

// State control
GVL_Machine.PackTags[UnitNo.Allocate].Command.CntrlCmd := ePMLCommand_Reset;
GVL_Machine.PackTags[UnitNo.Storage].Command.CntrlCmd := ePMLCommand_Reset;
GVL_Machine.PackTags[UnitNo.Shipping].Command.CntrlCmd := ePMLCommand_Reset;
arAxisCtrl_gb[AxisNo.RoundBelt].Admin.PositionType := E_PositionType.Modulo;
arAxisCtrl_gb[AxisNo.TurnTable].Admin.PositionType := E_PositionType.Modulo;

CASE eModeCurrent OF
    E_UnitMode.Manual:
        IF GVL_Machine.PackTags[UnitNo.Allocate].Status.StateCurrent = ePMLState_Idle AND
            GVL_Machine.PackTags[UnitNo.Storage].Status.StateCurrent = ePMLState_Idle AND
            GVL_Machine.PackTags[UnitNo.Shipping].Status.StateCurrent = ePMLState_Idle //
			 THEN
            M_StateComplete();
        END_IF
		IF ErrorTableInitDone THEN
			M_General_AlarmRegister();
		END_IF
    E_UnitMode.Auto:
        IF GVL_Machine.PackTags[UnitNo.Allocate].Status.StateCurrent = ePMLState_Idle AND
            GVL_Machine.PackTags[UnitNo.Storage].Status.StateCurrent = ePMLState_Idle AND
            GVL_Machine.PackTags[UnitNo.Shipping].Status.StateCurrent = ePMLState_Idle //AND
             THEN
            M_StateComplete();
        END_IF
		IF ErrorTableInitDone THEN
			M_General_AlarmRegister();
		END_IF
END_CASE
END_METHOD

METHOD M_RobotResetCmd : BOOL
VAR_INPUT
END_VAR
VAR
	bTrig : BOOL ;
END_VAR
bTrig := TRUE;

IF bTrig THEN
	RobotService_ResetCmd := TRUE;
	bTrig := FALSE;
END_IF

IF TON_RobotReleaseResetCmd.Q THEN
	RobotService_ResetCmd := FALSE;
	M_RobotResetCmd := TRUE;
END_IF
END_METHOD

METHOD M_RobotStartCmd : BOOL
VAR_INPUT
END_VAR
VAR
	bTrig	: BOOL;
END_VAR
bTrig := TRUE;

IF bTrig THEN
	RobotService_StartCmd := TRUE;
	bTrig := FALSE;
END_IF

IF TON_RobotReleaseStartCmd.Q THEN
	RobotService_StartCmd := FALSE;
	M_RobotStartCmd := TRUE;
END_IF
END_METHOD

METHOD M_ShippingRobotResetCmd : BOOL
VAR_INPUT
END_VAR

VAR
	bTrig: BOOL;
END_VAR
bTrig := TRUE;

IF bTrig THEN
	ShippingRobotService_ResetCmd := TRUE;
	bTrig := FALSE;
END_IF

IF TON_Shipping_RobotRelease_ResetCmd.Q THEN
	ShippingRobotService_ResetCmd := FALSE;
	M_ShippingRobotResetCmd := TRUE;
END_IF
END_METHOD

METHOD M_ShippingRobotStartCmd : BOOL
VAR_INPUT
END_VAR

VAR
	bTrig: BOOL;
END_VAR
bTrig := TRUE;

IF bTrig THEN
	ShippingRobotService_StartCmd := TRUE;
	bTrig := FALSE;
END_IF

IF TON_Shipping_RobotRelease_StartCmd.Q THEN
	ShippingRobotService_StartCmd := FALSE;
	M_ShippingRobotStartCmd := TRUE;
END_IF
END_METHOD

METHOD M_StartHoming
VAR_INPUT
END_VAR
fbMachineHoming.xExecute := TRUE;
END_METHOD

METHOD M_Starting
// State control
GVL_Machine.PackTags[UnitNo.Allocate].Command.CntrlCmd := ePMLCommand_Start;
GVL_Machine.PackTags[UnitNo.Storage].Command.CntrlCmd := ePMLCommand_Start;
GVL_Machine.PackTags[UnitNo.Shipping].Command.CntrlCmd := ePMLCommand_Start;

CASE eModeCurrent OF
    E_UnitMode.Manual, E_UnitMode.Auto:
        IF GVL_Machine.PackTags[UnitNo.Allocate].Status.StateCurrent = ePMLState_Execute AND
            GVL_Machine.PackTags[UnitNo.Allocate].Status.StateCurrent = ePMLState_Execute AND
            GVL_Machine.PackTags[UnitNo.Allocate].Status.StateCurrent = ePMLState_Execute THEN
            M_StateComplete();
        END_IF
END_CASE
END_METHOD

METHOD M_StopHoming
VAR_INPUT
END_VAR
fbMachineHoming.xExecute := FALSE;
END_METHOD

METHOD M_Stopped
VAR
	CylinderIndex : UDINT;
	MotorIndex : INT;
	ServoIndex : INT;
END_VAR
FOR ServoIndex := 1 TO 7 DO
	IF arAxisCtrl_gb[ServoIndex].Admin.Axis.Status.Error THEN
		arAxisCtrl_gb[ServoIndex].Admin.ClearError := FALSE;
	END_IF
END_FOR

IF eModeCurrent = E_UnitMode.Auto THEN
	GVL_Machine.PackTags[UnitNo.Storage].Command.UnitMode := E_UnitMode.Auto;
	GVL_Machine.PackTags[UnitNo.Allocate].Command.UnitMode := E_UnitMode.Auto;
	GVL_Machine.PackTags[UnitNo.Shipping].Command.UnitMode := E_UnitMode.Auto;
ELSIF eModeCurrent = E_UnitMode.Manual THEN
	GVL_Machine.PackTags[UnitNo.Storage].Command.UnitMode := E_UnitMode.Manual;
	GVL_Machine.PackTags[UnitNo.Allocate].Command.UnitMode := E_UnitMode.Manual;
	GVL_Machine.PackTags[UnitNo.Shipping].Command.UnitMode := E_UnitMode.Manual;
END_IF

CASE eModeCurrent OF
	E_UnitMode.Manual:
		IF GVL_Machine.PackTags[UnitNo.Allocate].Status.UnitModeCurrent = E_UnitMode.Manual AND 
			GVL_Machine.PackTags[UnitNo.Allocate].Status.StateCurrent = ePMLState_Stopped AND
			GVL_Machine.PackTags[UnitNo.Storage].Status.UnitModeCurrent = E_UnitMode.Manual AND 
			GVL_Machine.PackTags[UnitNo.Storage].Status.StateCurrent = ePMLState_Stopped AND
			GVL_Machine.PackTags[UnitNo.Shipping].Status.UnitModeCurrent = E_UnitMode.Manual AND 
			GVL_Machine.PackTags[UnitNo.Shipping].Status.StateCurrent = ePMLState_Stopped THEN
			M_StateComplete();
		END_IF
	E_UnitMode.Auto:
		IF GVL_Machine.PackTags[UnitNo.Allocate].Status.UnitModeCurrent = E_UnitMode.Auto AND 
			GVL_Machine.PackTags[UnitNo.Allocate].Status.StateCurrent = ePMLState_Stopped AND
			GVL_Machine.PackTags[UnitNo.Storage].Status.UnitModeCurrent = E_UnitMode.Auto AND 
			GVL_Machine.PackTags[UnitNo.Storage].Status.StateCurrent = ePMLState_Stopped AND
			GVL_Machine.PackTags[UnitNo.Shipping].Status.UnitModeCurrent = E_UnitMode.Auto AND 
			GVL_Machine.PackTags[UnitNo.Shipping].Status.StateCurrent = ePMLState_Stopped THEN
			M_StateComplete();
		END_IF
END_CASE
END_METHOD

METHOD M_Stopping
VAR
	CylinderIndex :UDINT;
	MotorIndex : INT;
END_VAR
CASE eModeCurrent OF
    E_UnitMode.Manual:
        GVL_Machine.PackTags[UnitNo.Allocate].Command.UnitMode := E_UnitMode.Manual;
        GVL_Machine.PackTags[UnitNo.Allocate].Command.CntrlCmd := ePMLCommand_Stop;
        GVL_Machine.PackTags[UnitNo.Storage].Command.UnitMode  := E_UnitMode.Manual;
        GVL_Machine.PackTags[UnitNo.Storage].Command.CntrlCmd  := ePMLCommand_Stop;
        GVL_Machine.PackTags[UnitNo.Shipping].Command.UnitMode := E_UnitMode.Manual;
        GVL_Machine.PackTags[UnitNo.Shipping].Command.CntrlCmd := ePMLCommand_Stop;
		FOR CylinderIndex := 1 TO udiMax_CylinderNum DO
			Cylinder.arCylinder[CylinderIndex].xEnable := FALSE;
		END_FOR
		FOR MotorIndex := 1 TO 26 DO
			Motor.arMotor[MotorIndex].xEnable := FALSE;
		END_FOR
		TableMove.xExecute := FALSE;
        IF GVL_Machine.PackTags[UnitNo.Allocate].Status.UnitModeCurrent = E_UnitMode.Manual AND
           GVL_Machine.PackTags[UnitNo.Allocate].Status.StateCurrent = ePMLState_Stopped AND
           GVL_Machine.PackTags[UnitNo.Storage].Status.UnitModeCurrent = E_UnitMode.Manual AND
           GVL_Machine.PackTags[UnitNo.Storage].Status.StateCurrent = ePMLState_Stopped AND
           GVL_Machine.PackTags[UnitNo.Shipping].Status.UnitModeCurrent = E_UnitMode.Manual AND
           GVL_Machine.PackTags[UnitNo.Shipping].Status.StateCurrent = ePMLState_Stopped AND NOT
		   TableMove.xError
            THEN
            M_StateComplete();
        END_IF
	E_UnitMode.Auto:
        GVL_Machine.PackTags[UnitNo.Allocate].Command.UnitMode := E_UnitMode.Auto;
        GVL_Machine.PackTags[UnitNo.Allocate].Command.CntrlCmd := ePMLCommand_Stop;
        GVL_Machine.PackTags[UnitNo.Storage].Command.UnitMode  := E_UnitMode.Auto;
        GVL_Machine.PackTags[UnitNo.Storage].Command.CntrlCmd  := ePMLCommand_Stop;
        GVL_Machine.PackTags[UnitNo.Shipping].Command.UnitMode := E_UnitMode.Auto;
        GVL_Machine.PackTags[UnitNo.Shipping].Command.CntrlCmd := ePMLCommand_Stop;
		FOR CylinderIndex := 1 TO udiMax_CylinderNum DO
			Cylinder.arCylinder[CylinderIndex].xEnable := FALSE;
		END_FOR
		FOR MotorIndex := 1 TO 26 DO
			Motor.arMotor[MotorIndex].xEnable := FALSE;
		END_FOR
		TableMove.xExecute := FALSE;
        IF GVL_Machine.PackTags[UnitNo.Allocate].Status.UnitModeCurrent = E_UnitMode.Auto AND
           GVL_Machine.PackTags[UnitNo.Allocate].Status.StateCurrent = ePMLState_Stopped AND
           GVL_Machine.PackTags[UnitNo.Storage].Status.UnitModeCurrent = E_UnitMode.Auto AND
           GVL_Machine.PackTags[UnitNo.Storage].Status.StateCurrent = ePMLState_Stopped AND
           GVL_Machine.PackTags[UnitNo.Shipping].Status.UnitModeCurrent = E_UnitMode.Auto AND
           GVL_Machine.PackTags[UnitNo.Shipping].Status.StateCurrent = ePMLState_Stopped AND NOT
		   TableMove.xError
            THEN
            M_StateComplete();
        END_IF
END_CASE
END_METHOD

METHOD PRIVATE M_StroageRobotSafeCheck : BOOL
VAR_INPUT
END_VAR
IF FanucRobot.List.StorageRobot._DI12.BzoneWaitAllow THEN
	IF NOT arAxisCtrl_gb[AxisNo.RoundBelt].Admin.Axis.Status.Moving
	    AND NOT fbAllocateArea.RoundBeltControl.xBusy
		AND NOT fbAllocateArea.RoundBeltControl.xError
		AND NOT fbAllocateArea.RoundBeltControl.xDone THEN
			FanucRobot.List.StorageRobot.Bzone_AllowWork := TRUE;
	END_IF
END_IF

IF NOT FanucRobot.List.StorageRobot._DI12.BzoneInWork 
	AND NOT FanucRobot.List.StorageRobot._DI12.BzoneWaitAllow THEN
	FanucRobot.List.StorageRobot.Bzone_AllowWork := FALSE	;
END_IF
END_METHOD

METHOD M_Suspended
M_StateComplete();
END_METHOD

METHOD M_Suspending
M_StateComplete();
END_METHOD

METHOD M_Undefined
CASE eModeCurrent OF
    E_UnitMode.Undefined:
		PackTag.Command.UnitMode := E_UnitMode.Manual;
		PackTag.Command.CntrlCmd := ePMLCommand_Abort;
		M_StateComplete();
END_CASE
END_METHOD

METHOD M_Unholding
M_StateComplete();
END_METHOD

METHOD M_Unsuspending
M_StateComplete();
END_METHOD

METHOD PRIVATE RefAllocateService
VAR_INPUT
END_VAR
AllocateService.AllocateMoveStructure 				REF= Service_Handshake.AllocateMoveStructure;
AllocateService.AllocateCircleMove 					REF= Service_Handshake.AllocateCircleMove;
AllocateService.TurnTableMove 						REF= Service_Handshake.TurnTableMove;

// Allocating
AllocateService.AutoMode_AllocateBatchMode 			REF= Service_Handshake.AutoMode_AllocateBatchMode;
AllocateService.AutoMode_SimpleAllocation_Batch 	REF= Service_Handshake.AutoMode_SimpleAllocation_Batch;
AllocateService.AutoMode_AllocateBatchMode_Reverse  REF= Service_Handshake.AutoMode_AllocateBatchMode_Reverse;

//OutRobot
AllocateService.AutoMode_RareBoxMove 				REF= Service_Handshake.AutoMode_RareBoxMove;
AllocateService.AutoMode_EmptyBoxMove 				REF= Service_Handshake.AutoMode_EmptyBoxMove;
AllocateService.AutoMode_BoxMoveReverse 			REF= Service_Handshake.AutoMode_BoxMoveReverse;

//TransCV camera 
AllocateService.AutoMode_SameSizeCVCamera 			REF= Service_Handshake.AutoMode_SameSizeCVCamera;
AllocateService.AutoMode_SameSizeCVCamera_Reverse 	REF= Service_Handshake.AutoMode_SameSizeCVCamera_Reverse;
AllocateService.AutoMode_DifferentCVCamera 			REF= Service_Handshake.AutoMode_DifferentCVCamera;

//AllocateArea Home
AllocateService.AllocateRegionHome					REF= Service_Handshake.AllocationRegionHome;

// Pullout 
AllocateService.AutoMode_PullOutConveyor 			REF= Service_Handshake.AutoMode_PullOutConveyor;

//AutoModeUse*-------自動模式圓帶單動
   AllocateService.AutoMode_AllocateCircleMove 		 REF= Service_Handshake.AutoMode_AllocateCircleMove;

 //AutoModeUse*-------圓盤移動
    AllocateService.AutoMode_TurnTableMOve  		REF= Service_Handshake.AutoMode_TurnTableMOve;
	
//Allocate robot move
AllocateService.AllocateRobotNeedlingMove 			REF= Service_Handshake.AllocationRobotNeedlingMove;

//逆向拍照批次入料
AllocateService.AutoMode_ReverseBatchPick			REF= Service_Handshake.AutoMode_ReverseBatchPick;

//同尺寸軌道回倉/NG
AllocateService.AutoMode_ReverseBoxToWareHouse		REF= Service_Handshake.AutoMode_ReverseBoxToWareHouse;
END_METHOD

